	        // ----------------------------------------->>>>>>> STATUS MANUAL <<<<<<<-----------------------------------------
	        
	        // Write to static from IO
	        // ACTIVATE --> MANUAL MODE
	        // ProductionLine
	        IF #Active.Line.ProductionLine THEN
	            // SET --> MANUAL MODE
	            IF DB_Manual.Line.ProductionLine.Conveyor[#ConveyorID].ManualEnable THEN
	                #ReadConveyorStatus.Manual := TRUE;
	            END_IF;
	            // RESET --> MANUAL MODE
	            IF NOT DB_Manual.Line.ProductionLine.Conveyor[#ConveyorID].ManualEnable AND #SSR.ResetSystem THEN
	                #ReadConveyorStatus.Manual := FALSE;
	            END_IF;
	        END_IF;
	        // EmptyLine
	        IF #Active.Line.EmptyLine THEN
	            // SET --> MANUAL MODE
	            IF DB_Manual.Line.EmptyLine.Conveyor[#ConveyorID].ManualEnable THEN
	                #ReadConveyorStatus.Manual := TRUE;
	            END_IF;
	            // RESET --> MANUAL MODE
	            IF NOT DB_Manual.Line.EmptyLine.Conveyor[#ConveyorID].ManualEnable AND #SSR.ResetSystem THEN
	                #ReadConveyorStatus.Manual := FALSE;
	            END_IF;
	        END_IF;
	        // PackedLine
	        IF #Active.Line.PackedLine THEN
	            // SET --> MANUAL MODE
	            IF DB_Manual.Line.PackedLine.Conveyor[#ConveyorID].ManualEnable THEN
	                #ReadConveyorStatus.Manual := TRUE;
	            END_IF;
	            // RESET --> MANUAL MODE
	            IF NOT DB_Manual.Line.PackedLine.Conveyor[#ConveyorID].ManualEnable AND #SSR.ResetSystem THEN
	                #ReadConveyorStatus.Manual := FALSE;
	            END_IF;
	        END_IF;
	        
	        // Manual enable and Run from HMI
	        // ProductionLine
	        IF #Active.Line.ProductionLine THEN
	            IF #ConveyorID = DB_Manual.Conveyor.ID THEN
	                DB_Manual.Line.ProductionLine.Conveyor[DB_Manual.Conveyor.ID].ManualEnable := DB_Manual.Conveyor.Enable;
	                DB_Manual.Line.ProductionLine.Conveyor[DB_Manual.Conveyor.ID].Run.Forward := DB_Manual.Conveyor.in;
	            END_IF;
	        END_IF;
	        // EmptyLine
	        IF #Active.Line.EmptyLine THEN
	            IF #ConveyorID = DB_Manual.Conveyor.ID THEN
	                DB_Manual.Line.EmptyLine.Conveyor[DB_Manual.Conveyor.ID].ManualEnable := DB_Manual.Conveyor.Enable;
	                DB_Manual.Line.EmptyLine.Conveyor[DB_Manual.Conveyor.ID].Run.Forward := DB_Manual.Conveyor.in;
	            END_IF;
	        END_IF;
	        // PackedLine
	        IF #Active.Line.PackedLine THEN
	            IF #ConveyorID = DB_Manual.Conveyor.ID THEN
	                DB_Manual.Line.PackedLine.Conveyor[DB_Manual.Conveyor.ID].ManualEnable := DB_Manual.Conveyor.Enable;
	                DB_Manual.Line.PackedLine.Conveyor[DB_Manual.Conveyor.ID].Run.Forward := DB_Manual.Conveyor.in;
	            END_IF;
	        END_IF;
	        
	    END_REGION
	    
	    REGION Status Stop
	        
	        // ----------------------------------------->>>>>>> STATUS STOP <<<<<<<-----------------------------------------
	        
	        IF #SSR.StopSystem THEN
	            #ReadConveyorStatus.Stop := TRUE;
	        END_IF;
	        IF #SSR.StartSystem OR #SSR.ResetSystem THEN
	            #ReadConveyorStatus.Stop := FALSE;
	        END_IF;
	        
	    END_REGION
	    
	    REGION Sensor Blockage
	        
	        // ----------------------------------------->>>>>>> STATUS BLOCKAGE <<<<<<<------------------------------------
	        
	        // FB_SensorBlockage
	        // called as MIDB
	        #CONVEYOR_SENSOR_BLOCKAGE(ConveyorSensor       := #FilteredSensor,
	                                  StatusRunning        := #ReadConveyorStatus.Running,
	                                  SensorBlockagePeriod := #ReadConveyorParameters.SensorBlockageTime,
	                                  SensorBlocked        => #ConveyorFault.Sensor_Blockage,
	                                  ReadBlockageStatus   => #ReadConveyorStatus.Blockage);
	        
	        REGION alarm 
	            
	            // ==========================
	            // Sensor Blockage: HMI Alarm
	            // ==========================
	            // Sensor blockage alarm message is written to the alarm word
	            // corresponding to the active line
	            // ProductionLine
	            IF #Active.Line.ProductionLine THEN
	                DB_Alarm."word".Line.ProductionLine.Conveyor[#ConveyorID].%X0 := #ReadConveyorStatus.Blockage;
	            END_IF;
	            // EmptyLine
	            IF #Active.Line.EmptyLine THEN
	                DB_Alarm."word".Line.EmptyLine.Conveyor[#ConveyorID].%X0 := #ReadConveyorStatus.Blockage;
	            END_IF;
	            // PackedLine
	            IF #Active.Line.PackedLine THEN
	                DB_Alarm."word".Line.PackedLine.Conveyor[#ConveyorID].%X0 := #ReadConveyorStatus.Blockage;
	            END_IF;
	            
	        END_REGION
	        
	    END_REGION
	    
	    REGION Visu Color
	        
	        // each and every status of the conveyor will be mentioned by different colors in HMI panel
	        
	        #VisuColor.%X8 := #ReadConveyorStatus.Blockage;
	        #VisuColor.%X0 := #ReadConveyorStatus.ON;
	        #VisuColor.%X1 := #ReadConveyorStatus.ReadytoRun;
	        #VisuColor.%X2 := #ReadConveyorStatus.Occupied;
	        #VisuColor.%X3 := #ReadConveyorStatus.Running;
	        #VisuColor.%X4 := #ReadConveyorStatus.Fault;
	        #VisuColor.%X5 := #ReadConveyorStatus.Estop;
	        #VisuColor.%X6 := #ReadConveyorStatus.Manual;
	        #VisuColor.%X7 := #ReadConveyorStatus.Stop;
	        
	        // convert word to Interger value: 
	        // color will be depends on the status priority (integer value) 
	        // reference: Conveyor image in HMI screen -> property -> Apperance   
	        
	        // ProductionLine
	        IF #Active.Line.ProductionLine THEN
	            DB_VisuColor.Line.ProductionLine.Conveyor[#ConveyorID] :=
	            WORD_TO_INT(#VisuColor);
	        END_IF;
	        // EmptyLine
	        IF #Active.Line.EmptyLine THEN
	            DB_VisuColor.Line.EmptyLine.Conveyor[#ConveyorID] :=
	            WORD_TO_INT(#VisuColor);
	        END_IF;
	        // PackedLine
	        IF #Active.Line.PackedLine THEN
	            DB_VisuColor.Line.PackedLine.Conveyor[#ConveyorID] :=
	            WORD_TO_INT(#VisuColor);
	        END_IF;
	        
	    END_REGION
	    
	    REGION Global Status
	        
	        // write -> global status
	        // ProductionLine
	        IF #Active.Line.ProductionLine THEN
	            DB_Global.Status.Line.ProductionLine.On[#ConveyorID] := #ReadConveyorStatus.ON;
	            DB_Global.Status.Line.ProductionLine.ReadyToRun[#ConveyorID] := #ReadConveyorStatus.ReadytoRun;
	            DB_Global.Status.Line.ProductionLine.Occupied[#ConveyorID] := #ReadConveyorStatus.Occupied;
	            DB_Global.Status.Line.ProductionLine.Running[#ConveyorID] := #ReadConveyorStatus.Running;
	            DB_Global.Status.Line.ProductionLine.Fault[#ConveyorID] := #ReadConveyorStatus.Fault;
	            DB_Global.Status.Line.ProductionLine.Estop[#ConveyorID] := #ReadConveyorStatus.Estop;
	            DB_Global.Status.Line.ProductionLine.Manual[#ConveyorID] := #ReadConveyorStatus.Manual;
	            DB_Global.Status.Line.ProductionLine.Stop[#ConveyorID] := #ReadConveyorStatus.Stop;
	            DB_Global.Status.Line.ProductionLine.Blockage[#ConveyorID] := #ReadConveyorStatus.Blockage;
	        END_IF;
	        // EmptyLine
	        IF #Active.Line.EmptyLine THEN
	            DB_Global.Status.Line.EmptyLine.On[#ConveyorID] := #ReadConveyorStatus.ON;
	            DB_Global.Status.Line.EmptyLine.ReadyToRun[#ConveyorID] := #ReadConveyorStatus.ReadytoRun;
	            DB_Global.Status.Line.EmptyLine.Occupied[#ConveyorID] := #ReadConveyorStatus.Occupied;
	            DB_Global.Status.Line.EmptyLine.Running[#ConveyorID] := #ReadConveyorStatus.Running;
	            DB_Global.Status.Line.EmptyLine.Fault[#ConveyorID] := #ReadConveyorStatus.Fault;
	            DB_Global.Status.Line.EmptyLine.Estop[#ConveyorID] := #ReadConveyorStatus.Estop;
	            DB_Global.Status.Line.EmptyLine.Manual[#ConveyorID] := #ReadConveyorStatus.Manual;
	            DB_Global.Status.Line.EmptyLine.Stop[#ConveyorID] := #ReadConveyorStatus.Stop;
	            DB_Global.Status.Line.EmptyLine.Blockage[#ConveyorID] := #ReadConveyorStatus.Blockage;
	        END_IF;
	        // PackedLine
	        IF #Active.Line.PackedLine THEN
	            DB_Global.Status.Line.PackedLine.On[#ConveyorID] := #ReadConveyorStatus.ON;
	            DB_Global.Status.Line.PackedLine.ReadyToRun[#ConveyorID] := #ReadConveyorStatus.ReadytoRun;
	            DB_Global.Status.Line.PackedLine.Occupied[#ConveyorID] := #ReadConveyorStatus.Occupied;
	            DB_Global.Status.Line.PackedLine.Running[#ConveyorID] := #ReadConveyorStatus.Running;
	            DB_Global.Status.Line.PackedLine.Fault[#ConveyorID] := #ReadConveyorStatus.Fault;
	            DB_Global.Status.Line.PackedLine.Estop[#ConveyorID] := #ReadConveyorStatus.Estop;
	            DB_Global.Status.Line.PackedLine.Manual[#ConveyorID] := #ReadConveyorStatus.Manual;
	            DB_Global.Status.Line.PackedLine.Stop[#ConveyorID] := #ReadConveyorStatus.Stop;
	            DB_Global.Status.Line.PackedLine.Blockage[#ConveyorID] := #ReadConveyorStatus.Blockage;
	        END_IF;
	        
	    END_REGION
	    
	END_REGION
	
	REGION Run/Stop Conveyor 
	    
	    // FB_ConveyorRunStop
	    // Called as MIDB
	    
	    #"RUN/STOP_CONVEYOR"(StatusReady  := #ReadConveyorStatus.ReadytoRun,
	                         StatusOccu   := #ReadConveyorStatus.Occupied,
	                         DSOcc        := #Downstream,
	                         USOcc        := #Upstream,
	                         EnergySave   := #EnergySave,
	                         ILStop       := #Interlock,
	                         PecBlockage  := #ConveyorFault.Sensor_Blockage,
	                         MotorForward => #StartMotorForward,
	                         MotorReverse => #StartMotorReverse);
	    
	END_REGION
	
	REGION Energy Save
	    
	    // FB_EnergySave
	    // Called as MIDB
	    
	    #ENERGY_SAVE(StatusReady      := #ReadConveyorStatus.ReadytoRun,
	                 StatusOccupied   := #ReadConveyorStatus.Occupied,
	                 StartUpIN        := #SetStartUp,
	                 USOcc            := #Upstream,
	                 EnergySaveTimePT := #ReadConveyorParameters.EnergySaveTime,
	                 EnergySaveOut    => #EnergySave);
	    
	END_REGION
	
	REGION Write logic and parameters
	    
	    // Motor Forward: motors which has only one control bit
	    // ProductionLine 
	    IF #Active.Line.ProductionLine THEN
	        #RunForward :=
	        (#StartMotorForward AND NOT #StartMotorReverse) // Automatic mode
	        OR (#ReadConveyorStatus.Manual AND DB_Manual.Line.ProductionLine.Conveyor[#ConveyorID].Run.Forward); //Manual mode
	    END_IF;
	    // EmptyLine 
	    IF #Active.Line.EmptyLine THEN
	        #RunForward :=
	        (#StartMotorForward AND NOT #StartMotorReverse) // Automatic mode
	        OR (#ReadConveyorStatus.Manual AND DB_Manual.Line.EmptyLine.Conveyor[#ConveyorID].Run.Forward); //Manual mode
	    END_IF;
	    // PackedLine 
	    IF #Active.Line.PackedLine THEN
	        #RunForward :=
	        (#StartMotorForward AND NOT #StartMotorReverse) // Automatic mode
	        OR (#ReadConveyorStatus.Manual AND DB_Manual.Line.PackedLine.Conveyor[#ConveyorID].Run.Forward); //Manual mode
	    END_IF;
	    
	    REGION Bihl Wiedemann 
	        
	        // process data for BW-ASi
	        
	        IF #MotorType."24v-ASi" THEN
	            
	            REGION Direction
	                
	                // ProductionLine
	                IF #Active.Line.ProductionLine THEN
	                    #WriteAsiDir := DB_AsiSetpoint.Line.ProductionLine.DirChange.Conveyor[#ConveyorID];
	                END_IF;
	                // EmptyLine
	                IF #Active.Line.EmptyLine THEN
	                    #WriteAsiDir := DB_AsiSetpoint.Line.EmptyLine.DirChange.Conveyor[#ConveyorID];
	                END_IF;
	                // PackedLine
	                IF #Active.Line.PackedLine THEN
	                    #WriteAsiDir := DB_AsiSetpoint.Line.PackedLine.DirChange.Conveyor[#ConveyorID];
	                END_IF;
	                
	            END_REGION
	            
	            REGION Speed
	                
	                // ProductionLine
	                IF #Active.Line.ProductionLine THEN
	                    #WriteAsiSpeed := DB_AsiSetpoint.Line.ProductionLine.Speed.Conveyor[#ConveyorID];
	                END_IF;
	                // EmptyLine
	                IF #Active.Line.EmptyLine THEN
	                    #WriteAsiSpeed := DB_AsiSetpoint.Line.EmptyLine.Speed.Conveyor[#ConveyorID];
	                END_IF;
	                // PackedLine
	                IF #Active.Line.PackedLine THEN
	                    #WriteAsiSpeed := DB_AsiSetpoint.Line.PackedLine.Speed.Conveyor[#ConveyorID];
	                END_IF;
	                
	            END_REGION
	            
	        END_IF;
	        
	    END_REGION
	    
	    REGION NORD (Line shaft)
	        
	        // process data and logic for NORD VFD
	        
	        IF #MotorType.nord THEN
	            
	            // ProductionLine
	            IF #Active.Line.ProductionLine THEN
	                
	                IF NOT #ReadConveyorStatus.Fault THEN
	                    IF // Nord Motor Run - Automatic mode
	                        ((#ReadConveyorStatus.ReadytoRun AND
	                        #StartMotorForward) OR
	                        // Nord Motor Run - manual mode
	                        (#ReadConveyorStatus.Manual AND
	                        DB_Manual.Line.ProductionLine.Conveyor[#ConveyorID].Run.Forward))
	                    THEN
	                        #NordControlEnable := #NordSetpointRun;
	                    ELSE
	                        #NordControlEnable := #NordSetpointReady;
	                    END_IF;
	                END_IF;
	                
	                // Nord Motor Fault ack
	                IF #ReadConveyorStatus.Fault AND #SSR.ResetSystem THEN
	                    #NordControlEnable := #NordFaultAck;
	                END_IF;
	                
	                // Nord setpoint
	                #NordSetpoint := DINT_TO_WORD(DB_NordSetPoint.Line.ProductionLine.Conveyor[#ConveyorID]);
	                
	            END_IF;
	            
	            // EmptyLine
	            IF #Active.Line.EmptyLine THEN
	                
	                IF NOT #ReadConveyorStatus.Fault THEN
	                    IF // Nord Motor Run - Automatic mode
	                        ((#ReadConveyorStatus.ReadytoRun AND
	                        #StartMotorForward) OR
	                        // Nord Motor Run - manual mode
	                        (#ReadConveyorStatus.Manual AND
	                        DB_Manual.Line.EmptyLine.Conveyor[#ConveyorID].Run.Forward))
	                    THEN
	                        #NordControlEnable := #NordSetpointRun;
	                    ELSE
	                        #NordControlEnable := #NordSetpointReady;
	                    END_IF;
	                END_IF;
	                
	                // Nord Motor Fault ack
	                IF #ReadConveyorStatus.Fault AND #SSR.ResetSystem THEN
	                    #NordControlEnable := #NordFaultAck;
	                END_IF;
	                
	                // Nord setpoint
	                #NordSetpoint := DINT_TO_WORD(DB_NordSetPoint.Line.EmptyLine.Conveyor[#ConveyorID]);
	                
	            END_IF;
	            
	            // PackedLine
	            IF #Active.Line.PackedLine THEN
	                
	                IF NOT #ReadConveyorStatus.Fault THEN
	                    IF // Nord Motor Run - Automatic mode
	                        ((#ReadConveyorStatus.ReadytoRun AND
	                        #StartMotorForward) OR
	                        // Nord Motor Run - manual mode
	                        (#ReadConveyorStatus.Manual AND
	                        DB_Manual.Line.PackedLine.Conveyor[#ConveyorID].Run.Forward))
	                    THEN
	                        #NordControlEnable := #NordSetpointRun;
	                    ELSE
	                        #NordControlEnable := #NordSetpointReady;
	                    END_IF;
	                END_IF;
	                
	                // Nord Motor Fault ack
	                IF #ReadConveyorStatus.Fault AND #SSR.ResetSystem THEN
	                    #NordControlEnable := #NordFaultAck;
	                END_IF;
	                
	                // Nord setpoint
	                #NordSetpoint := DINT_TO_WORD(DB_NordSetPoint.Line.PackedLine.Conveyor[#ConveyorID]);
	                
	            END_IF;
	            
	            
	   END_IF;
	            
	            
	END_REGION
	
	REGION Interroll Multi control roller
	    
	    // process data for Interroll multicontrol card
	    IF #MotorType."24v-IMC" THEN
	    // PackedLine
	        IF #Active.Line.PackedLine THEN
	            IF (#StartMotorForward AND NOT #StartMotorReverse)
	            OR (#ReadConveyorStatus.Manual AND
	            DB_Manual.Line.PackedLine.Conveyor[#ConveyorID].Run.Forward AND
	            NOT DB_Manual.Line.PackedLine.Conveyor[#ConveyorID].Run.Reverse)
	           THEN
	            #ImcSpeed := #ReadConveyorParameters."IMC-SpeedSetPoint";
	           ELSE
	            #ImcSpeed := #NullSpeed;
	           END_IF;
	       END_IF;
	   END_IF;
	   
	END_REGION
	    
	END_REGION
	
END_FUNCTION_BLOCK
END_NAMESPACE

NAMESPACE Global
FUNCTION_BLOCK FB_MABS
{ S7_Optimized_Access := 'TRUE' ; Published := 'TRUE' }
VERSION : 0.1
   VAR_INPUT 
      MABS_ID : Int;
      CrossSensor : Bool;
      ErrorSignal : Bool;
      Upstream : Bool;
      UpstreamRunning : Bool;
      Downstream_Straight : Bool;
      "Downstream_Right/Left" : Bool;
      SortDir : ItemDir;
      RemoteOut1 : Bool;
      RemoteOut2 : Bool;
      RemoteOut3 : Bool;
      RemoteOut4 : Bool;
      Parameter : MABS_Parameters;
   END_VAR

   VAR_OUTPUT 
      RemoteIn1 : Bool;
      RemoteIn2 : Bool;
      RemoteIn3 : Bool;
      RunWheels : Bool;
   END_VAR

   VAR 
      ReadInputSignal : Struct
         CrossSensor : Bool;
         EmergencyStop : Bool;
         ErrorSignal : Bool;
      END_STRUCT;
      Active : Struct
         Line : Struct
            ProductionLine : Bool;
            EmptyLine : Bool;
            PackedLine : Bool;
         END_STRUCT;
         EstopZone { S7_SetPoint := 'False'} : EsopZone;
      END_STRUCT;
      CROSS_SENSOR_FILTER { S7_SetPoint := 'False'} : FB_Sensor;
      MABS_SENSOR_BLOCKAGE {InstructionName := 'IEC_TIMER'; LibVersion := '1.0'} : IEC_TIMER;
      MABS_STATUS_ON { S7_SetPoint := 'False'} : FB_StatusON;
      MABS_STATUS_READY { S7_SetPoint := 'False'} : FB_StatusReady;
      MABS_STATUS_FAULT { S7_SetPoint := 'False'} : FB_StatusFault;
      AUTO_RESET { S7_SetPoint := 'False'} : FB_AutoReset;
      SSR { S7_SetPoint := 'False'} : SystemSSR;
      ReadMabsStatus { S7_SetPoint := 'False'} : ConveyorStatus;
      MABSFault { S7_SetPoint := 'False'} : Fault;
      SimuMode : Struct
         Sensor : Bool;
         Fault : Bool;
      END_STRUCT;
      StartUpTimer {InstructionName := 'TOF_TIME'; LibVersion := '1.0'; S7_SetPoint := 'False'} : TOF_TIME;
      FT_StartUp {InstructionName := 'F_TRIG'; LibVersion := '1.0'} : F_TRIG;
      SetStartUp { S7_SetPoint := 'True'} : Bool;
      VisuColor : Word;
      PhaseError : Bool;
      StartupMABS { S7_SetPoint := 'True'} : Bool;
      FilteredSensor { S7_SetPoint := 'True'} : Bool;
      AutoReset { S7_SetPoint := 'True'} : Bool;
      StopSystemFireActive : Bool;
      Sort { S7_SetPoint := 'False'} : ItemDir;
      mabs : Struct
         RemoteIn1 : Bool;
         RemoteIn2 : Bool;
         RemoteIn3 : Bool;
         RemoteIn4 : Bool;
         Wheels : Bool;
      END_STRUCT;
      Home : Bool;
      HomeCheckTimer {InstructionName := 'TON_TIME'; LibVersion := '1.0'} : TON_TIME;
      CurrentPosition : Struct
         left : Bool;
         right : Bool;
         straight : Bool;
      END_STRUCT;
      RT_DelaySwing_Straight {InstructionName := 'R_TRIG'; LibVersion := '1.0'} : R_TRIG;
      RT_DelaySwing_toRight {InstructionName := 'R_TRIG'; LibVersion := '1.0'} : R_TRIG;
      RT_DelaySwing_toLeft {InstructionName := 'R_TRIG'; LibVersion := '1.0'} : R_TRIG;
      ToSt_DelayTimer {InstructionName := 'TON_TIME'; LibVersion := '1.0'} : TON_TIME;
      ToRt_DelayTimer {InstructionName := 'TON_TIME'; LibVersion := '1.0'} : TON_TIME;
      ToLt_DelayTimer {InstructionName := 'TON_TIME'; LibVersion := '1.0'} : TON_TIME;
      St_SwingDelay { S7_SetPoint := 'True'} : Bool;
      Rt_SwingDelay : Bool;
      Lt_SwingDelay : Bool;
      noSwing : Bool;
      CmdExFailure : Struct
         "Timer" {InstructionName := 'TONR_TIME'; LibVersion := '1.0'} : TONR_TIME;
         UpstreamCheckTimer {InstructionName := 'TONR_TIME'; LibVersion := '1.0'} : TONR_TIME;
      END_STRUCT;
      FT_Upstream {InstructionName := 'F_TRIG'; LibVersion := '1.0'; S7_SetPoint := 'False'} : F_TRIG;
      RT_DS_St {InstructionName := 'R_TRIG'; LibVersion := '1.0'} : R_TRIG;
      "RT_DS_Rt/Lt" {InstructionName := 'R_TRIG'; LibVersion := '1.0'} : R_TRIG;
      RT_ToStraight {InstructionName := 'R_TRIG'; LibVersion := '1.0'; S7_SetPoint := 'False'} : R_TRIG;
      RT_ToRight {InstructionName := 'R_TRIG'; LibVersion := '1.0'} : R_TRIG;
      RT_ToLeft {InstructionName := 'R_TRIG'; LibVersion := '1.0'} : R_TRIG;
      FT_Blockage {InstructionName := 'F_TRIG'; LibVersion := '1.0'} : F_TRIG;
      HoldFailure { S7_SetPoint := 'True'} : Bool;
      MABS_Wheel {InstructionName := 'TOF_TIME'; LibVersion := '1.0'; S7_SetPoint := 'False'} : TOF_TIME;
      RT_Sort_St {InstructionName := 'R_TRIG'; LibVersion := '1.0'} : R_TRIG;
      RT_Sort_Rt {InstructionName := 'R_TRIG'; LibVersion := '1.0'} : R_TRIG;
      RT_Sort_Lt {InstructionName := 'R_TRIG'; LibVersion := '1.0'} : R_TRIG;
      HoldSwingTimer {InstructionName := 'TOF_TIME'; LibVersion := '1.0'} : TOF_TIME;
      HoldSwing { S7_SetPoint := 'True'} : Bool;
   END_VAR


BEGIN
	// ==========================================================================================================================================
	// Company        : LogTech, s.r.o.
	// Created by     : Anton Vinoth Soundraraj
	// Block          : FB_MABS
	// Project        : Lékarna DC Chrudim
	// Project number : 23-157
	// ==========================================================================================================================================
	
	REGION Active Line
	    
	    // ProductionLine
	    IF (#MABS_ID >= _.gminProductionLine AND
	        #MABS_ID <= _.gmaxProductionLine)
	    THEN
	        #Active.Line.ProductionLine := TRUE;
	    END_IF;
	    
	    // EmptyLine
	    IF (#MABS_ID >= _.gminEmptyLine AND
	        #MABS_ID <= _.gmaxEmptyLine)
	    THEN
	        #Active.Line.EmptyLine := TRUE;
	    END_IF;
	    
	    // PackedLine
	    IF (#MABS_ID >= _.gminPackedLine AND
	        #MABS_ID <= _.gmaxPackedLine)
	    THEN
	        #Active.Line.PackedLine := TRUE;
	    END_IF;
	    
	END_REGION
	    
	
	REGION Estop zone
	    
	    // Production Line A1
	    IF (#MABS_ID >= _."gA1.6.1" AND
	        #MABS_ID <= _."gA1.6.2") OR
	        // Empty Line A1
	        (#MABS_ID >= _."gJ1.5.2" AND
	        #MABS_ID <= _."gJ1.6.2")
	    THEN
	        #Active.EstopZone."1" := TRUE;
	    END_IF;
	    
	    // Production Line A2
	    IF (#MABS_ID >= _."gA1.9.1" AND
	        #MABS_ID <= _."gA1.9.2")
	    THEN
	        #Active.EstopZone."2" := TRUE;
	    END_IF;
	    
	END_REGION
	
	REGION Read Simu inputs  
	    
	    // ProductionLine
	    IF #Active.Line.ProductionLine THEN
	        // read simu
	        #SimuMode.Sensor := DB_SystemSimu.TriggerSensor.Line.ProductionLine.Conveyor[#MABS_ID];
	        #SimuMode.Fault := DB_SystemSimu.TriggerFault.Line.ProductionLine.Conveyor[#MABS_ID];
	    END_IF;
	    
	    // EmptyLine
	    IF #Active.Line.EmptyLine THEN
	        // read simu
	        #SimuMode.Sensor := DB_SystemSimu.TriggerSensor.Line.EmptyLine.Conveyor[#MABS_ID];
	        #SimuMode.Fault := DB_SystemSimu.TriggerFault.Line.EmptyLine.Conveyor[#MABS_ID];
	    END_IF;
	    
	    // PackedLine
	    IF #Active.Line.PackedLine THEN
	        // read simu
	        #SimuMode.Sensor := DB_SystemSimu.TriggerSensor.Line.PackedLine.Conveyor[#MABS_ID];
	        #SimuMode.Fault := DB_SystemSimu.TriggerFault.Line.PackedLine.Conveyor[#MABS_ID];
	    END_IF;
	    
	END_REGION
	
	REGION SystemSSR
	    
	    //Zone 1
	    IF #Active.EstopZone."1" THEN
	        #SSR.StartSystem := DB_SystemSSR.Zone."1".StartSystem;
	        #SSR.StopSystem := DB_SystemSSR.Zone."1".StopSystem;
	        #SSR.ResetSystem := DB_SystemSSR.Zone."1".ResetSystem;
	    END_IF;
	    
	    //Zone 2
	    IF #Active.EstopZone."2" THEN
	        #SSR.StartSystem := DB_SystemSSR.Zone."2".StartSystem;
	        #SSR.StopSystem := DB_SystemSSR.Zone."2".StopSystem;
	        #SSR.ResetSystem := DB_SystemSSR.Zone."2".ResetSystem;
	    END_IF;
	    
	END_REGION
	
	REGION Read Input
	    
	    // read all inputs to the block
	    // Conveyor input read signals
	    #ReadInputSignal.CrossSensor := #CrossSensor OR
	    #SimuMode.Sensor; // simu call
	    #ReadInputSignal.ErrorSignal := #ErrorSignal OR
	    #SimuMode.Fault; // simu call;
	    // estop
	    #ReadInputSignal.EmergencyStop := _.DB_SafetyStandard.ToStandard.EstopActive;
	    
	END_REGION
	
	REGION Conveyor startup
	    
	    // Conveyor StartUp: Conveyor startup signal after 5 second delay
	    
	    #StartUpTimer.TOF(IN := #SSR.StartSystem,
	                      PT := #Parameter.StartUpTime);
	    
	    #FT_StartUp(CLK := #StartUpTimer.Q);
	    
	    // set startup after 5 seconds
	    #SetStartUp := #FT_StartUp.Q;
	    
	END_REGION
	
	REGION READ AND INIT
	    
	    REGION FIRE
	        
	        // Fire signal from fire system stops the whole system
	        // System can be reset from Fire status only if the fire signal is deactivated
	        
	        // FIRE ALARM ACTIVE --> STOP SYSTEM
	        IF DB_SystemSimu.Fire THEN
	            #StopSystemFireActive := TRUE;
	        END_IF;
	        // RESET --> FIRE ALARM
	        IF #SSR.ResetSystem AND NOT DB_SystemSimu.Fire THEN
	            #StopSystemFireActive := FALSE;
	        END_IF;
	        
	    END_REGION
	    
	END_REGION
	
	REGION Conveyor Status
	    
	    REGION Status ON
	        
	        // ----------------------------------------->>>>>>> STATUS ON <<<<<<<-----------------------------------------
	        // FB_ConveyorStatusON
	        // called as IDMB
	        
	        #MABS_STATUS_ON(SystemStartActive := #SSR.StartSystem,
	                        StatusStop := #ReadMabsStatus.Stop,
	                        StatusEStop := #ReadMabsStatus.Estop,
	                        StatusManual := #ReadMabsStatus.Manual,
	                        StatusFault := #ReadMabsStatus.Fault,
	                        FireAlarmActive := #StopSystemFireActive,
	                        StatusON => #ReadMabsStatus.ON);
	        
	    END_REGION
	    
	    REGION Status Ready
	        
	        // ----------------------------------------->>>>>>> STATUS READY <<<<<<<-----------------------------------------
	        // FB_ConveyorStatusReady
	        // called as MIDB
	        
	        #MABS_STATUS_READY(StatusON := #ReadMabsStatus.ON,
	                           StatusESTOP := #ReadMabsStatus.Estop,
	                           StatusFAULT := #ReadMabsStatus.Fault,
	                           StatusMAN := #ReadMabsStatus.Manual,
	                           SignalFIRE := #StopSystemFireActive,
	                           SystemAlertTime := #Parameter.StartUpTime,
	                           StatusReady => #ReadMabsStatus.ReadytoRun);
	        
	    END_REGION
	    
	    REGION Status Occupied
	        
	        // ----------------------------------------->>>>>>> STATUS OCCUPIED <<<<<<<-----------------------------------------
	        
	        #ReadMabsStatus.Occupied :=
	        #CROSS_SENSOR_FILTER.FilteredSensor;
	        
	    END_REGION
	    
	    REGION Status Running
	        
	        // ----------------------------------------->>>>>>> STATUS RUNNING <<<<<<<-----------------------------------------
	        
	        #ReadMabsStatus.Running :=
	        #ReadMabsStatus.ReadytoRun AND
	        #mabs.Wheels;
	        
	    END_REGION
	    
	    REGION Status Fault
	        
	        // ----------------------------------------->>>>>>> STATUS FAULT <<<<<<<-----------------------------------------
	        
	        // Reading error signal from the motor drive
	        #MABSFault.Motor_Error := #ReadInputSignal.ErrorSignal;
	        
	        // FC_ConveyorStatusFault
	        #MABS_STATUS_FAULT(FaultActive := #MABSFault.Motor_Error,
	                           ResetFault := #SSR.ResetSystem,
	                           StatusRunning := #ReadMabsStatus.Running,
	                           FaultStatus => #ReadMabsStatus.Fault);
	        
	    END_REGION
	    
	    REGION Status ESTOP
	        
	        // ----------------------------------------->>>>>>> STATUS ESTOP <<<<<<<-----------------------------------------
	        
	        #AUTO_RESET(AckIN := #SSR.ResetSystem,
	                    Ack => #AutoReset);
	        
	        // EMERGENCY STOP ACTIVE --> STOP SYSTEM
	        IF #ReadInputSignal.EmergencyStop THEN
	            #ReadMabsStatus.Estop := TRUE;
	        END_IF;
	        // RESET --> EMERGENCY STOP
	        IF #AutoReset AND NOT #ReadInputSignal.EmergencyStop THEN
	            #ReadMabsStatus.Estop := FALSE;
	        END_IF;
	        
	    END_REGION
	    
	    REGION Status Stop
	        
	        // ----------------------------------------->>>>>>> STATUS STOP <<<<<<<-----------------------------------------
	        
	        IF #SSR.StopSystem THEN
	            #ReadMabsStatus.Stop := TRUE;
	        END_IF;
	        IF #SSR.StartSystem OR #SSR.ResetSystem THEN
	            #ReadMabsStatus.Stop := FALSE;
	        END_IF;
	        
	    END_REGION
	    
	    REGION Sensor Blockage
	        
	        // ----------------------------------------->>>>>>> STATUS BLOCKAGE <<<<<<<-------------------------------------
	        
	        // FB_SensorBlockage
	        // called as MIDB
	        
	        #MABS_SENSOR_BLOCKAGE.TON(IN := #ReadMabsStatus.ReadytoRun AND
	                                  #CROSS_SENSOR_FILTER.FilteredSensor,
	                                  PT := #Parameter.SensorBlockageTime,
	                                  Q => #ReadMabsStatus.Blockage);
	        
	        // ==========================
	        // Sensor Blockage: HMI Alarm
	        // ==========================
	        // Sensor blockage alarm message is written to the first bit of the alarm word
	        // corresponding to the active line
	        
	        REGION alarm 
	            
	            // ==========================
	            // Sensor Blockage: HMI Alarm
	            // ==========================
	            // Sensor blockage alarm message is written to the alarm word
	            // corresponding to the active line
	            // ProductionLine
	            IF #Active.Line.ProductionLine THEN
	                DB_Alarm."word".Line.ProductionLine.Conveyor[#MABS_ID].%X0 := #ReadMabsStatus.Blockage;
	            END_IF;
	            // EmptyLine
	            IF #Active.Line.EmptyLine THEN
	                DB_Alarm."word".Line.EmptyLine.Conveyor[#MABS_ID].%X0 := #ReadMabsStatus.Blockage;
	            END_IF;
	            // PackedLine
	            IF #Active.Line.PackedLine THEN
	                DB_Alarm."word".Line.PackedLine.Conveyor[#MABS_ID].%X0 := #ReadMabsStatus.Blockage;
	            END_IF;
	            
	        END_REGION
	        
	    END_REGION
	    
	    REGION Global Status
	        
	        // write -> global status
	        // ProductionLine
	        IF #Active.Line.ProductionLine THEN
	            DB_Global.Status.Line.ProductionLine.On[#MABS_ID] := #ReadMabsStatus.ON;
	            DB_Global.Status.Line.ProductionLine.ReadyToRun[#MABS_ID] := #ReadMabsStatus.ReadytoRun;
	            DB_Global.Status.Line.ProductionLine.Occupied[#MABS_ID] := #ReadMabsStatus.Occupied;
	            DB_Global.Status.Line.ProductionLine.Running[#MABS_ID] := #ReadMabsStatus.Running;
	            DB_Global.Status.Line.ProductionLine.Fault[#MABS_ID] := #ReadMabsStatus.Fault;
	            DB_Global.Status.Line.ProductionLine.Estop[#MABS_ID] := #ReadMabsStatus.Estop;
	            DB_Global.Status.Line.ProductionLine.Manual[#MABS_ID] := #ReadMabsStatus.Manual;
	            DB_Global.Status.Line.ProductionLine.Stop[#MABS_ID] := #ReadMabsStatus.Stop;
	            DB_Global.Status.Line.ProductionLine.Blockage[#MABS_ID] := #ReadMabsStatus.Blockage;
	        END_IF;
	        // EmptyLine
	        IF #Active.Line.EmptyLine THEN
	            DB_Global.Status.Line.EmptyLine.On[#MABS_ID] := #ReadMabsStatus.ON;
	            DB_Global.Status.Line.EmptyLine.ReadyToRun[#MABS_ID] := #ReadMabsStatus.ReadytoRun;
	            DB_Global.Status.Line.EmptyLine.Occupied[#MABS_ID] := #ReadMabsStatus.Occupied;
	            DB_Global.Status.Line.EmptyLine.Running[#MABS_ID] := #ReadMabsStatus.Running;
	            DB_Global.Status.Line.EmptyLine.Fault[#MABS_ID] := #ReadMabsStatus.Fault;
	            DB_Global.Status.Line.EmptyLine.Estop[#MABS_ID] := #ReadMabsStatus.Estop;
	            DB_Global.Status.Line.EmptyLine.Manual[#MABS_ID] := #ReadMabsStatus.Manual;
	            DB_Global.Status.Line.EmptyLine.Stop[#MABS_ID] := #ReadMabsStatus.Stop;
	            DB_Global.Status.Line.EmptyLine.Blockage[#MABS_ID] := #ReadMabsStatus.Blockage;
	        END_IF;
	        // PackedLine
	        IF #Active.Line.PackedLine THEN
	            DB_Global.Status.Line.PackedLine.On[#MABS_ID] := #ReadMabsStatus.ON;
	            DB_Global.Status.Line.PackedLine.ReadyToRun[#MABS_ID] := #ReadMabsStatus.ReadytoRun;
	            DB_Global.Status.Line.PackedLine.Occupied[#MABS_ID] := #ReadMabsStatus.Occupied;
	            DB_Global.Status.Line.PackedLine.Running[#MABS_ID] := #ReadMabsStatus.Running;
	            DB_Global.Status.Line.PackedLine.Fault[#MABS_ID] := #ReadMabsStatus.Fault;
	            DB_Global.Status.Line.PackedLine.Estop[#MABS_ID] := #ReadMabsStatus.Estop;
	            DB_Global.Status.Line.PackedLine.Manual[#MABS_ID] := #ReadMabsStatus.Manual;
	            DB_Global.Status.Line.PackedLine.Stop[#MABS_ID] := #ReadMabsStatus.Stop;
	            DB_Global.Status.Line.PackedLine.Blockage[#MABS_ID] := #ReadMabsStatus.Blockage;
	        END_IF;
	        
	    END_REGION
	    
	    REGION Visu Color
	        
	        // each and every status of the conveyor will be mentioned by different colors in HMI panel
	        
	        #VisuColor.%X8 := #ReadMabsStatus.Blockage;
	        #VisuColor.%X0 := #ReadMabsStatus.ON;
	        #VisuColor.%X1 := #ReadMabsStatus.ReadytoRun;
	        #VisuColor.%X2 := #ReadMabsStatus.Occupied;
	        #VisuColor.%X3 := #ReadMabsStatus.Running;
	        #VisuColor.%X4 := #ReadMabsStatus.Fault;
	        #VisuColor.%X5 := #ReadMabsStatus.Estop;
	        #VisuColor.%X6 := #ReadMabsStatus.Manual;
	        #VisuColor.%X7 := #ReadMabsStatus.Stop;
	        
	        // convert word to Interger value: 
	        // color will be depends on the status priority (integer value) 
	        // reference: Conveyor image in HMI screen -> property -> Apperance   
	        
	        // ProductionLine
	        IF #Active.Line.ProductionLine THEN
	            DB_VisuColor.Line.ProductionLine.Conveyor[#MABS_ID] :=
	            WORD_TO_INT(#VisuColor);
	        END_IF;
	        // EmptyLine
	        IF #Active.Line.EmptyLine THEN
	            DB_VisuColor.Line.EmptyLine.Conveyor[#MABS_ID] :=
	            WORD_TO_INT(#VisuColor);
	        END_IF;
	        // PackedLine
	        IF #Active.Line.PackedLine THEN
	            DB_VisuColor.Line.PackedLine.Conveyor[#MABS_ID] :=
	            WORD_TO_INT(#VisuColor);
	        END_IF;
	        
	    END_REGION
	    
	END_REGION
	
	REGION Sorter sensor filter
	    
	    // cross sensor filter
	    #CROSS_SENSOR_FILTER(Sensor := #ReadInputSignal.CrossSensor,   ///#CrossSensor
	                         SensorFilterTime := #Parameter.CrossSensorFilterTime);
	    
	    
	END_REGION
	
	REGION MABS FUNCTIONALITY
	    
	    REGION rcv direction 
	        
	(*        // only if the mabs is not performing any operation
	        IF NOT #Upstream
	        THEN
	            #HoldSwing := TRUE;
	        ELSE
	            #HoldSwing := FALSE;
	        END_IF;
	        
	        IF NOT #HoldSwing THEN
	            
	            #Sort := #SortDir;
	            
	        END_IF; *)
	        
	        #Sort := #SortDir;
	        
	    END_REGION
	    
	    // Signal to RemoteIN1 / RemoteIN2 for specify swing direction and RemoteIN3 for swing must be 50ms or longer.
	    // Otherwise transfer ball may behaves unexpectedly.
	    // If the signal input of IN1 and IN2 (specifying the swing direction) is delayed from the signal input of IN3 (swing RUN),
	    // an unintended swing operation will occur.
	    // After outputting the swinging status, turn RemoteIN3 (Swing start) OFF.
	    
	    REGION MABS wheels
	        
	        // run mobs wheel 
	        // runs only when remoteIn3(swing) not active
	        
	        #mabs.Wheels := #UpstreamRunning;
	        
	    END_REGION
	    
	    // ==========================================================================================================================
	    // Swing status output
	    // ===================
	    
	    // SWING STATUS         RemoteOUT2  RemoteOUT3   Remark
	    // ------------         ----------  ----------   ------
	    // Straight (origin)        ON          ON       Outputs at the time when balls have been turned to the straight direction.
	    // Swing (CW)               ON          OFF      Outputs at the time when swing in CW direction is complete.
	    // Swing (CCW)              OFF         ON       Outputs at the time when swing in CCW direction is complete.
	    // Others                   OFF         OFF      During ball swing, when turning on power supply,
	    //                                               undetected swing position or occurring software error.
	    // ==========================================================================================================================                                              
	    
	    REGION Current position
	        
	        // current MABS position
	        
	        #CurrentPosition.left :=
	        NOT #RemoteOut2 AND
	        #RemoteOut3;
	        
	        #CurrentPosition.right :=
	        #RemoteOut2 AND
	        NOT #RemoteOut3;
	        
	        #CurrentPosition.straight :=
	        #RemoteOut2 AND
	        #RemoteOut3;
	        
	    END_REGION
	    
	    REGION HOMING
	        
	        // ==========================================================================================================================
	        // Initial operation (origin searching)
	        // ===================================
	        
	        #HomeCheckTimer.TON(IN := NOT #CurrentPosition.left AND
	                            NOT #CurrentPosition.right AND
	                            NOT #CurrentPosition.straight,
	                            PT := T#1s);
	        
	        #Home :=
	        NOT #HomeCheckTimer.Q;
	        
	        // home missing
	        
	        IF NOT #Home AND NOT #ReadMabsStatus.Stop THEN
	            #mabs.RemoteIn1 := TRUE;
	            #mabs.RemoteIn2 := TRUE;
	            #mabs.RemoteIn3 := TRUE;
	        END_IF;
	        
	    END_REGION
	    
	    // ==========================================================================================================================
	    // Specified swing direction
	    // =========================
	    
	    // SWING                                                    RemoteIN1  RemoteIN2   
	    // -----                                                    ---------  ---------   
	    // Divert direction to Straight direction (CW direction)       ON          ON       
	    // Divert direction to Straight direction (CCW direction)      ON          OFF      
	    // Straight direction to Divert direction (CW direction)       OFF         ON       
	    // Straight direction to Divert direction (CCW direction)      OFF         OFF                                                    .
	    // ==========================================================================================================================
	    // Start swinging
	    // ==============
	    
	    // swing    RemoteIN3
	    // -----    ---------  
	    // STOP         OFF
	    // RUN          ON  .
	    
	    // ==========================================================================================================================
	    
	    IF #ReadMabsStatus.ReadytoRun AND NOT #HoldFailure
	    THEN
	        
	        REGION swing delay
	            
	            #ToSt_DelayTimer(IN := #mabs.#RemoteIn1 AND #mabs.#RemoteIn2,
	                             PT := t#20ms,
	                             Q => #St_SwingDelay);
	            
	            #ToRt_DelayTimer(IN := NOT #mabs.#RemoteIn1 AND #mabs.#RemoteIn2,
	                             PT := t#20ms,
	                             Q => #Rt_SwingDelay);
	            
	            #ToLt_DelayTimer(IN := #mabs.#RemoteIn1 AND NOT #mabs.#RemoteIn2,
	                             PT := t#20ms,
	                             Q => #Lt_SwingDelay);
	            
	            // swing starts after few ms of turn decision made
	            IF (#St_SwingDelay OR
	                #Rt_SwingDelay OR
	                #Lt_SwingDelay) AND
	                NOT #noSwing
	            THEN
	                #mabs.RemoteIn3 := TRUE;
	            END_IF;
	            
	        END_REGION
	        
	        REGION Straight
	            
	            IF (#CurrentPosition.straight AND
	                #Sort.Straight) OR
	                (#CurrentPosition.right AND
	                #Sort.toRight) OR
	                (#CurrentPosition.left AND
	                #Sort.toLeft)
	            THEN
	                #mabs.RemoteIn3 := FALSE;
	                #noSwing := TRUE;
	            ELSE
	                #noSwing := FALSE;
	            END_IF;
	            
	            
	            // ================================================== ^^^
	            
	            // sort straight - actual position: right
	            
	            IF #Sort.Straight AND
	                NOT #CurrentPosition.straight AND
	                #CurrentPosition.right AND
	                NOT #CROSS_SENSOR_FILTER.FilteredSensor
	            THEN
	                #mabs.#RemoteIn1 := TRUE;
	                #mabs.RemoteIn2 := TRUE;
	            END_IF;
	            
	            // sort straight - actual position: left
	            
	            IF #Sort.Straight AND
	                NOT #CurrentPosition.straight AND
	                #CurrentPosition.left AND
	                NOT #CROSS_SENSOR_FILTER.FilteredSensor
	            THEN
	                #mabs.#RemoteIn1 := TRUE;
	                #mabs.RemoteIn2 := TRUE;
	            END_IF;
	            
	            // sort straight - actual position: straight
	            
	            IF #Sort.Straight AND
	                #CurrentPosition.straight AND
	                NOT #CurrentPosition.left AND
	                NOT #CurrentPosition.right AND
	                NOT #CROSS_SENSOR_FILTER.FilteredSensor
	            THEN
	                #mabs.RemoteIn3 := FALSE; // no swing
	            END_IF;
	            
	        END_REGION
	        
	        REGION to Right
	            
	            #RT_DelaySwing_toRight(CLK := #ToRt_DelayTimer.Q);
	            
	            // ================================================== >>>
	            
	            // sort right - actual position: straight/left
	            
	            IF #Sort.toRight AND
	                NOT #CurrentPosition.right AND
	                (#CurrentPosition.straight OR
	                #CurrentPosition.left) AND
	                NOT #CROSS_SENSOR_FILTER.FilteredSensor
	            THEN
	                #mabs.#RemoteIn1 := FALSE;
	                #mabs.RemoteIn2 := TRUE;
	            END_IF;
	            
	            // sort right - actual position: right
	            
	            IF #Sort.toRight AND
	                #CurrentPosition.right AND
	                NOT #CurrentPosition.left AND
	                NOT #CurrentPosition.straight AND
	                NOT #CROSS_SENSOR_FILTER.FilteredSensor
	            THEN
	                #mabs.RemoteIn3 := FALSE; // no swing
	            END_IF;
	            
	        END_REGION
	        
	        REGION to left
	            
	            #RT_DelaySwing_toLeft(CLK := #ToLt_DelayTimer.Q);
	            
	            // ================================================== <<<
	            
	            // sort left - actual position: straight/right
	            
	            IF #Sort.toLeft AND
	                NOT #CurrentPosition.left AND
	                (#CurrentPosition.straight OR
	                #CurrentPosition.right) AND
	                NOT #CROSS_SENSOR_FILTER.FilteredSensor
	            THEN
	                #mabs.#RemoteIn1 := FALSE;
	                #mabs.RemoteIn2 := TRUE;
	            END_IF;
	            
	            // sort left - actual position: left
	            
	            IF #Sort.toLeft AND
	                #CurrentPosition.left AND
	                NOT #CurrentPosition.straight AND
	                NOT #CurrentPosition.right AND
	                NOT #CROSS_SENSOR_FILTER.FilteredSensor
	            THEN
	                #mabs.RemoteIn3 := FALSE; // no swing
	            END_IF;
	            
	        END_REGION
	        
	        // ============================================================================================================
	        
	        #RemoteIn1 := #mabs.RemoteIn1;
	        #RemoteIn2 := #mabs.RemoteIn2;
	        #RemoteIn3 := #mabs.RemoteIn3;
	        
	        #RunWheels := #mabs.Wheels;
	        
	    END_IF;
	    
	    REGION Cmd excecution failure
	        
	        // if the cmd could not be excecuted, MABS getting program reset automatically
	        // Hold failure: makes all output to MABS value 0
	        // then starts executing cmd again
	        
	        IF #ReadMabsStatus.ReadytoRun AND #Home THEN
	            
	            // reset state change
	            #FT_Upstream(CLK := #Upstream);
	            #RT_DS_St(CLK := #Downstream_Straight);
	            #"RT_DS_Rt/Lt"(CLK := #"Downstream_Right/Left");
	            
	            // upstream not able to send tote in to MABS
	            #CmdExFailure.UpstreamCheckTimer(IN := #Upstream AND
	                                             ((NOT #Downstream_Straight AND #Sort.Straight) OR
	                                             (NOT #"Downstream_Right/Left" AND #Sort.toLeft)),
	                                             R := (#CmdExFailure.UpstreamCheckTimer.ET > t#30s) OR
	                                             #FT_Upstream.Q OR
	                                             #RT_DS_St.Q OR
	                                             #"RT_DS_Rt/Lt".Q OR
	                                             #SSR.ResetSystem,
	                                             PT := t#24h);
	            
	            // reset state change
	            #RT_ToStraight(CLK := #CurrentPosition.straight);
	            #RT_ToRight(CLK := #CurrentPosition.right);
	            #RT_ToLeft(CLK := #CurrentPosition.left);
	            #FT_Blockage(CLK := #ReadMabsStatus.Blockage);
	            
	            #CmdExFailure.Timer(IN := ((#Sort.Straight AND
	                                NOT #CurrentPosition.straight) OR
	                                (#Sort.toRight AND
	                                NOT #CurrentPosition.right) OR
	                                (#Sort.toLeft AND
	                                NOT #CurrentPosition.left)) OR
	                                #ReadMabsStatus.Blockage,
	                                R := (#CmdExFailure.Timer.ET > t#10s) OR
	                                #RT_ToStraight.Q OR
	                                #RT_ToRight.Q OR
	                                #RT_ToLeft.Q OR
	                                #FT_Blockage.Q OR
	                                #SSR.ResetSystem,
	                                PT := t#24h);
	            
	            #HoldFailure :=
	            ((#CmdExFailure.Timer.ET > t#5s) OR
	            (#CmdExFailure.UpstreamCheckTimer.ET > t#15s));
	            
	        END_IF;
	        
	        
	    END_REGION
	    
	    // stop if not ready
	    IF #Home AND (NOT #ReadMabsStatus.ReadytoRun OR #HoldFailure)
	    THEN
	        #RemoteIn1 := FALSE;
	        #RemoteIn2 := FALSE;
	        #RemoteIn3 := FALSE;
	        #RunWheels := FALSE;
	    END_IF;
	    
	    IF NOT #Home THEN
	        
	        #RemoteIn1 := #mabs.RemoteIn1;
	        #RemoteIn2 := #mabs.RemoteIn2;
	        #RemoteIn3 := #mabs.RemoteIn3;
	        
	    END_IF;
	    
	    
	END_REGION
	
	
	
END_FUNCTION_BLOCK
END_NAMESPACE

NAMESPACE Global
FUNCTION_BLOCK FB_MABS_Profinet
{ S7_Optimized_Access := 'TRUE' ; Published := 'TRUE' }
VERSION : 0.1
   VAR_INPUT 
      MABS_ID : Int;
      CrossSensor : Bool;
      Fault : Bool;
      UpstreamRunning : Bool;
      Downstream_Straight : Bool;
      "Downstream_Right/Left" : Bool;
      SortDir : ItemDir;
      ManIn : MABS_ManIn;
      Setpoints : MABS_Setpoint;
   END_VAR

   VAR_IN_OUT 
      MABS_IBP_in : IB_P01_02_03_in_64bytes_struct;
      MABS_IBP_out : IB_P01_02_03_out_64bytes_struct;
   END_VAR

   VAR 
      ReadInputSignal : Struct
         CrossSensor : Bool;
         EmergencyStop : Bool;
         Fault : Bool;
      END_STRUCT;
      Active : Struct
         Line : Struct
            ProductionLine : Bool;
            EmptyLine : Bool;
            PackedLine : Bool;
         END_STRUCT;
         EstopZone { S7_SetPoint := 'False'} : EsopZone;
      END_STRUCT;
      CROSS_SENSOR_FILTER : FB_Sensor;
      MABS_SENSOR_BLOCKAGE {InstructionName := 'IEC_TIMER'; LibVersion := '1.0'} : IEC_TIMER;
      MABS_STATUS_ON : FB_StatusON;
      MABS_STATUS_READY : FB_StatusReady;
      MABS_STATUS_FAULT : FB_StatusFault;
      AUTO_RESET : FB_AutoReset;
      MABS_CONTROL : FB_MABS_PNIO;
      SSR : SystemSSR;
      ReadMabsStatus : ConveyorStatus;
      ReadMabsParameter : ConveyorParameters := ((), [2(T#10ms)], (), (), (), ());
      MABSFault : Fault;
      SimuMode : Struct
         Sensor : Bool;
         Fault : Bool;
      END_STRUCT;
      StartUpTimer {InstructionName := 'TOF_TIME'; LibVersion := '1.0'; S7_SetPoint := 'False'} : TOF_TIME;
      FT_StartUp {InstructionName := 'F_TRIG'; LibVersion := '1.0'} : F_TRIG;
      SetStartUp { S7_SetPoint := 'True'} : Bool;
      VisuColor : Word;
      PhaseError : Bool;
      StartupMABS { S7_SetPoint := 'True'} : Bool;
      FilteredSensor { S7_SetPoint := 'True'} : Bool;
      AutoReset { S7_SetPoint := 'True'} : Bool;
      StopSystemFireActive : Bool;
      Sort { S7_SetPoint := 'False'} : ItemDir;
      Home : Bool;
      HomeCheckTimer {InstructionName := 'TON_TIME'; LibVersion := '1.0'} : TON_TIME;
      CurrentPosition : Struct
         left : Bool;
         right : Bool;
         straight : Bool;
      END_STRUCT;
      "Cmd+Setpoint" { ExternalAccessible := 'False'; ExternalVisible := 'False'; ExternalWritable := 'False'; S7_SetPoint := 'False'} : MABS;
   END_VAR


BEGIN
	// ==========================================================================================================================================
	// Company        : LogTech, s.r.o.
	// Created by     : Anton Vinoth Soundraraj
	// Block          : FB_MABS
	// Project        : Lékarna DC Chrudim
	// Project number : 23-157
	// ==========================================================================================================================================
	
	REGION Active Line
	    
	    // ProductionLine
	    IF (#MABS_ID >= _.gminProductionLine AND
	        #MABS_ID <= _.gmaxProductionLine)
	    THEN
	        #Active.Line.ProductionLine := TRUE;
	    END_IF;
	    
	    // EmptyLine
	    IF (#MABS_ID >= _.gminEmptyLine AND
	        #MABS_ID <= _.gmaxEmptyLine)
	    THEN
	        #Active.Line.EmptyLine := TRUE;
	    END_IF;
	    
	    // PackedLine
	    IF (#MABS_ID >= _.gminPackedLine AND
	        #MABS_ID <= _.gmaxPackedLine)
	    THEN
	        #Active.Line.PackedLine := TRUE;
	    END_IF;
	    
	END_REGION
	
	REGION Estop zone
	    
	    // Production Line A1
	    IF  (#MABS_ID >= _."gA1.6.1" AND
	        #MABS_ID <= _."gA1.6.2") OR
	        // Empty Line A1
	        (#MABS_ID >= _."gJ1.5.2" AND
	        #MABS_ID <= _."gJ1.6.2")
	    THEN
	        #Active.EstopZone."1" := TRUE;
	    END_IF;
	    
	    // Production Line A2
	    IF  (#MABS_ID >= _."gA1.9.1" AND
	        #MABS_ID <= _."gA1.9.2")
	    THEN
	        #Active.EstopZone."2" := TRUE;
	    END_IF;
	    
	END_REGION
	
	REGION SystemSSR
	    
	    //Zone 1
	    IF #Active.EstopZone."1" THEN
	        #SSR.StartSystem := DB_SystemSSR.Zone."1".StartSystem;
	        #SSR.StopSystem := DB_SystemSSR.Zone."1".StopSystem;
	        #SSR.ResetSystem := DB_SystemSSR.Zone."1".ResetSystem;
	    END_IF;
	    
	    //Zone 2
	    IF #Active.EstopZone."2" THEN
	        #SSR.StartSystem := DB_SystemSSR.Zone."2".StartSystem;
	        #SSR.StopSystem := DB_SystemSSR.Zone."2".StopSystem;
	        #SSR.ResetSystem := DB_SystemSSR.Zone."2".ResetSystem;
	    END_IF;
	    
	END_REGION
	
	REGION Read Simu inputs  
	    
	    // ProductionLine
	    IF #Active.Line.ProductionLine THEN
	        // read simu
	        #SimuMode.Sensor := DB_SystemSimu.TriggerSensor.Line.ProductionLine.Conveyor[#MABS_ID];
	        #SimuMode.Fault := DB_SystemSimu.TriggerFault.Line.ProductionLine.Conveyor[#MABS_ID];
	    END_IF;
	    
	    // EmptyLine
	    IF #Active.Line.EmptyLine THEN
	        // read simu
	        #SimuMode.Sensor := DB_SystemSimu.TriggerSensor.Line.EmptyLine.Conveyor[#MABS_ID];
	        #SimuMode.Fault := DB_SystemSimu.TriggerFault.Line.EmptyLine.Conveyor[#MABS_ID];
	    END_IF;
	    
	    // PackedLine
	    IF #Active.Line.PackedLine THEN
	        // read simu
	        #SimuMode.Sensor := DB_SystemSimu.TriggerSensor.Line.PackedLine.Conveyor[#MABS_ID];
	        #SimuMode.Fault := DB_SystemSimu.TriggerFault.Line.PackedLine.Conveyor[#MABS_ID];
	    END_IF;
	    
	END_REGION
	
	REGION Read Input
	    
	    // read all inputs to the block
	    // Conveyor input read signals
	    #ReadInputSignal.CrossSensor := #CrossSensor OR  // Not
	    #SimuMode.Sensor; // simu call
	    #ReadInputSignal.Fault := #Fault OR
	    #SimuMode.Fault; // simu call;
	    #ReadInputSignal.EmergencyStop := // all estop zones are connected together
	    _.DB_SafetyStandard.ToStandard.EstopActive;
	    
	END_REGION
	
	REGION READ AND INIT
	    
	    REGION parameters
	        
	        // ProductionLine
	        IF #Active.Line.ProductionLine THEN
	            #ReadMabsParameter := DB_ConveyorParameters.Line.ProductionLine.Conveyor[#MABS_ID];
	        END_IF;
	        // EmptyLine
	        IF #Active.Line.EmptyLine THEN
	            #ReadMabsParameter := DB_ConveyorParameters.Line.EmptyLine.Conveyor[#MABS_ID];
	        END_IF;
	        // PackedLine
	        IF #Active.Line.PackedLine THEN
	            #ReadMabsParameter := DB_ConveyorParameters.Line.PackedLine.Conveyor[#MABS_ID];
	        END_IF;
	        
	    END_REGION
	    
	    REGION FIRE
	        
	        // Fire signal from fire system stops the whole system
	        // System can be reset from Fire status only if the fire signal is deactivated
	        
	        // FIRE ALARM ACTIVE --> STOP SYSTEM
	        IF DB_SystemSimu.Fire THEN
	            #StopSystemFireActive := TRUE;
	        END_IF;
	        // RESET --> FIRE ALARM
	        IF #SSR.ResetSystem AND NOT DB_SystemSimu.Fire THEN
	            #StopSystemFireActive := FALSE;
	        END_IF;
	        
	    END_REGION
	    
	END_REGION
	
	REGION Conveyor startup
	    
	    // Conveyor StartUp: Conveyor startup signal after 5 second delay
	    
	    #StartUpTimer.TOF(IN := #SSR.StartSystem,
	                      PT := #ReadMabsParameter.StartUpTime);
	    
	    #FT_StartUp(CLK := #StartUpTimer.Q);
	    
	    // set startup after 5 seconds
	    #SetStartUp := #FT_StartUp.Q;
	    
	END_REGION
	
	REGION Conveyor Status
	    
	    REGION Status ON
	        
	        // ----------------------------------------->>>>>>> STATUS ON <<<<<<<-----------------------------------------
	        // FB_ConveyorStatusON
	        // called as IDMB
	        
	        #MABS_STATUS_ON(SystemStartActive := #SSR.StartSystem,
	                        StatusStop := #ReadMabsStatus.Stop,
	                        StatusEStop := #ReadMabsStatus.Estop,
	                        StatusManual := #ReadMabsStatus.Manual,
	                        StatusFault := #ReadMabsStatus.Fault,
	                        FireAlarmActive := #StopSystemFireActive,
	                        StatusON => #ReadMabsStatus.ON);
	        
	    END_REGION
	    
	    REGION Status Ready
	        
	        // ----------------------------------------->>>>>>> STATUS READY <<<<<<<-----------------------------------------
	        // FB_ConveyorStatusReady
	        // called as MIDB
	        
	        #MABS_STATUS_READY(StatusON := #ReadMabsStatus.ON,
	                           StatusESTOP := #ReadMabsStatus.Estop,
	                           StatusFAULT := #ReadMabsStatus.Fault,
	                           StatusMAN := #ReadMabsStatus.Manual,
	                           SignalFIRE := #StopSystemFireActive,
	                           SystemAlertTime := #ReadMabsParameter.StartUpTime,
	                           StatusReady => #ReadMabsStatus.ReadytoRun);
	        
	    END_REGION
	    
	    REGION Status Occupied
	        
	        // ----------------------------------------->>>>>>> STATUS OCCUPIED <<<<<<<-----------------------------------------
	        
	        #ReadMabsStatus.Occupied :=
	        #CROSS_SENSOR_FILTER.FilteredSensor;
	        
	    END_REGION
	    
	    REGION Status Running
	        
	        // ----------------------------------------->>>>>>> STATUS RUNNING <<<<<<<-----------------------------------------
	        
	        #ReadMabsStatus.Running :=
	        #ReadMabsStatus.ReadytoRun AND
	        #"Cmd+Setpoint".Run_balls;
	        
	    END_REGION
	    
	    REGION Status Fault
	        
	        // ----------------------------------------->>>>>>> STATUS FAULT <<<<<<<-----------------------------------------
	        
	        // Reading error signal from the motor drive
	        #MABSFault.Motor_Error := #ReadInputSignal.Fault;
	        
	        // FC_ConveyorStatusFault
	        #MABS_STATUS_FAULT(FaultActive := #MABSFault.Motor_Error,
	                           ResetFault := #SSR.ResetSystem,
	                           StatusRunning := #ReadMabsStatus.Running,
	                           FaultStatus => #ReadMabsStatus.Fault);
	        
	    END_REGION
	    
	    REGION Status ESTOP
	        
	        // ----------------------------------------->>>>>>> STATUS ESTOP <<<<<<<-----------------------------------------
	        
	        #AUTO_RESET(AckIN := #SSR.ResetSystem,
	                    Ack => #AutoReset);
	        
	        // EMERGENCY STOP ACTIVE --> STOP SYSTEM
	        IF #ReadInputSignal.EmergencyStop THEN
	            #ReadMabsStatus.Estop := TRUE;
	        END_IF;
	        // RESET --> EMERGENCY STOP
	        IF #AutoReset AND NOT #ReadInputSignal.EmergencyStop THEN
	            #ReadMabsStatus.Estop := FALSE;
	        END_IF;
	        
	    END_REGION
	    
	    REGION Status Stop
	        
	        // ----------------------------------------->>>>>>> STATUS STOP <<<<<<<-----------------------------------------
	        
	        IF #SSR.StopSystem THEN
	            #ReadMabsStatus.Stop := TRUE;
	        END_IF;
	        IF #SSR.StartSystem OR #SSR.ResetSystem THEN
	            #ReadMabsStatus.Stop := FALSE;
	        END_IF;
	        
	    END_REGION
	    
	    REGION Sensor Blockage
	        
	        // ----------------------------------------->>>>>>> STATUS BLOCKAGE <<<<<<<-------------------------------------
	        
	        // FB_SensorBlockage
	        // called as MIDB
	        
	        #MABS_SENSOR_BLOCKAGE.TON(IN := #ReadMabsStatus.ReadytoRun AND
	                                  #CROSS_SENSOR_FILTER.FilteredSensor,
	                                  PT := #ReadMabsParameter.SensorBlockageTime,
	                                  Q => #ReadMabsStatus.Blockage);
	        
	        // ==========================
	        // Sensor Blockage: HMI Alarm
	        // ==========================
	        // Sensor blockage alarm message is written to the first bit of the alarm word
	        // corresponding to the active line
	        
	        REGION alarm 
	            
	            // ==========================
	            // Sensor Blockage: HMI Alarm
	            // ==========================
	            // Sensor blockage alarm message is written to the alarm word
	            // corresponding to the active line
	            // ProductionLine
	            IF #Active.Line.ProductionLine THEN
	                DB_Alarm."word".Line.ProductionLine.Conveyor[#MABS_ID].%X0 := #ReadMabsStatus.Blockage;
	            END_IF;
	            // EmptyLine
	            IF #Active.Line.EmptyLine THEN
	               DB_Alarm."word".Line.EmptyLine.Conveyor[#MABS_ID].%X0 := #ReadMabsStatus.Blockage;
	            END_IF;
	            // PackedLine
	            IF #Active.Line.PackedLine THEN
	               DB_Alarm."word".Line.PackedLine.Conveyor[#MABS_ID].%X0 := #ReadMabsStatus.Blockage;
	            END_IF;
	            
	        END_REGION
	        
	    END_REGION
	    
	    REGION Visu Color
	        
	        // each and every status of the conveyor will be mentioned by different colors in HMI panel
	        
	        #VisuColor.%X8 := #ReadMabsStatus.Blockage;
	        #VisuColor.%X0 := #ReadMabsStatus.ON;
	        #VisuColor.%X1 := #ReadMabsStatus.ReadytoRun;
	        #VisuColor.%X2 := #ReadMabsStatus.Occupied;
	        #VisuColor.%X3 := #ReadMabsStatus.Running;
	        #VisuColor.%X4 := #ReadMabsStatus.Fault;
	        #VisuColor.%X5 := #ReadMabsStatus.Estop;
	        #VisuColor.%X6 := #ReadMabsStatus.Manual;
	        #VisuColor.%X7 := #ReadMabsStatus.Stop;
	        
	        // convert word to Interger value: 
	        // color will be depends on the status priority (integer value) 
	        // reference: Conveyor image in HMI screen -> property -> Apperance   
	        
	        // ProductionLine
	        IF #Active.Line.ProductionLine THEN
	            DB_VisuColor.Line.ProductionLine.Conveyor[#MABS_ID] :=
	            WORD_TO_INT(#VisuColor);
	        END_IF;
	        // EmptyLine
	        IF #Active.Line.EmptyLine THEN
	            DB_VisuColor.Line.EmptyLine.Conveyor[#MABS_ID] :=
	            WORD_TO_INT(#VisuColor);
	        END_IF;
	        // PackedLine
	        IF #Active.Line.PackedLine THEN
	            DB_VisuColor.Line.PackedLine.Conveyor[#MABS_ID] :=
	            WORD_TO_INT(#VisuColor);
	        END_IF;
	        
	    END_REGION
	    
	    REGION Global Status
	        
	        // write -> global status
	        // ProductionLine
	        IF #Active.Line.ProductionLine THEN
	            DB_Global.Status.Line.ProductionLine.On[#MABS_ID] := #ReadMabsStatus.ON;
	            DB_Global.Status.Line.ProductionLine.ReadyToRun[#MABS_ID] := #ReadMabsStatus.ReadytoRun;
	            DB_Global.Status.Line.ProductionLine.Occupied[#MABS_ID] := #ReadMabsStatus.Occupied;
	            DB_Global.Status.Line.ProductionLine.Running[#MABS_ID] := #ReadMabsStatus.Running;
	            DB_Global.Status.Line.ProductionLine.Fault[#MABS_ID] := #ReadMabsStatus.Fault;
	            DB_Global.Status.Line.ProductionLine.Estop[#MABS_ID] := #ReadMabsStatus.Estop;
	            DB_Global.Status.Line.ProductionLine.Manual[#MABS_ID] := #ReadMabsStatus.Manual;
	            DB_Global.Status.Line.ProductionLine.Stop[#MABS_ID] := #ReadMabsStatus.Stop;
	            DB_Global.Status.Line.ProductionLine.Blockage[#MABS_ID] := #ReadMabsStatus.Blockage;
	        END_IF;
	        // EmptyLine
	        IF #Active.Line.EmptyLine THEN
	            DB_Global.Status.Line.EmptyLine.On[#MABS_ID] := #ReadMabsStatus.ON;
	            DB_Global.Status.Line.EmptyLine.ReadyToRun[#MABS_ID] := #ReadMabsStatus.ReadytoRun;
	            DB_Global.Status.Line.EmptyLine.Occupied[#MABS_ID] := #ReadMabsStatus.Occupied;
	            DB_Global.Status.Line.EmptyLine.Running[#MABS_ID] := #ReadMabsStatus.Running;
	            DB_Global.Status.Line.EmptyLine.Fault[#MABS_ID] := #ReadMabsStatus.Fault;
	            DB_Global.Status.Line.EmptyLine.Estop[#MABS_ID] := #ReadMabsStatus.Estop;
	            DB_Global.Status.Line.EmptyLine.Manual[#MABS_ID] := #ReadMabsStatus.Manual;
	            DB_Global.Status.Line.EmptyLine.Stop[#MABS_ID] := #ReadMabsStatus.Stop;
	            DB_Global.Status.Line.EmptyLine.Blockage[#MABS_ID] := #ReadMabsStatus.Blockage;
	        END_IF;
	        // PackedLine
	        IF #Active.Line.PackedLine THEN
	            DB_Global.Status.Line.PackedLine.On[#MABS_ID] := #ReadMabsStatus.ON;
	            DB_Global.Status.Line.PackedLine.ReadyToRun[#MABS_ID] := #ReadMabsStatus.ReadytoRun;
	            DB_Global.Status.Line.PackedLine.Occupied[#MABS_ID] := #ReadMabsStatus.Occupied;
	            DB_Global.Status.Line.PackedLine.Running[#MABS_ID] := #ReadMabsStatus.Running;
	            DB_Global.Status.Line.PackedLine.Fault[#MABS_ID] := #ReadMabsStatus.Fault;
	            DB_Global.Status.Line.PackedLine.Estop[#MABS_ID] := #ReadMabsStatus.Estop;
	            DB_Global.Status.Line.PackedLine.Manual[#MABS_ID] := #ReadMabsStatus.Manual;
	            DB_Global.Status.Line.PackedLine.Stop[#MABS_ID] := #ReadMabsStatus.Stop;
	            DB_Global.Status.Line.PackedLine.Blockage[#MABS_ID] := #ReadMabsStatus.Blockage;
	        END_IF;
	        
	    END_REGION
	    
	END_REGION
	
	REGION Sorter sensor filter
	    
	    // cross sensor filter
	    #CROSS_SENSOR_FILTER(Sensor :=  #ReadInputSignal.CrossSensor,   ///#CrossSensor
	                         SensorFilterTime := #ReadMabsParameter.SensorFilterTime,
	                         FilteredSensor=> #FilteredSensor);
	    
	END_REGION
	
	REGION MABS LOGIC
	    
	    REGION rcv direction 
	        
	        IF NOT #FilteredSensor THEN
	            #Sort := #SortDir;
	        END_IF;
	        
	    END_REGION
	    
	    REGION MABS lib block
	        
	        #MABS_CONTROL(IBP_in  := #MABS_IBP_in,
	                      IBP_out := #MABS_IBP_out,
	                      MABS    := #"Cmd+Setpoint");
	        
	    END_REGION
	    
	    REGION run MABS wheels
	        
	        #"Cmd+Setpoint".Run_balls := #UpstreamRunning;
	        
	    END_REGION
	    
	    REGION Current position
	        
	        #CurrentPosition.left := #"Cmd+Setpoint".Left_Pos_reach;
	        #CurrentPosition.right := #"Cmd+Setpoint".Right_Pos_reach;
	        #CurrentPosition.straight := #"Cmd+Setpoint".Straight_Pos_reach;
	        
	    END_REGION
	    
	    REGION HOMING
	        
	        // ==========================================================================================================================
	        // Initial operation (home searching)
	        // ==================================
	        
	        // Home missing (if MABS could not receive any position in 't' duration)
	        #HomeCheckTimer.TON(IN := NOT #CurrentPosition.left AND
	                            NOT #CurrentPosition.right AND
	                            NOT #CurrentPosition.straight,
	                            PT := T#2s);
	        #Home :=
	        NOT #HomeCheckTimer.Q;
	        
	        // init HOME
	        IF NOT #Home AND NOT #ReadMabsStatus.Stop THEN
	            #"Cmd+Setpoint".Init := TRUE;
	        END_IF;
	        // RESET -> Init Home
	        IF #Home THEN
	            #"Cmd+Setpoint".Init := TRUE;
	        END_IF;
	        
	    END_REGION
	    
	    REGION Parameters
	        
	        // change balls direction
	        #"Cmd+Setpoint".Dir_balls := #Setpoints.ChangeBallsDirection;
	        // balls speed
	        #"Cmd+Setpoint".Speed_balls := #Setpoints.Speed_balls;
	        // offset for straight
	        #"Cmd+Setpoint".Init_offset := #Setpoints.Init_offset;
	        
	    END_REGION
	    
	    REGION Sorting logic
	        
	        IF #ReadMabsStatus.ReadytoRun
	        THEN
	            
	            REGION Straight
	                
	                // ================================================== ^^^
	                
	                // sort straight - actual position: right
	                
	                IF #Sort.Straight AND
	                    NOT #CurrentPosition.straight AND
	                    #CurrentPosition.right AND
	                    NOT #CROSS_SENSOR_FILTER.FilteredSensor
	                THEN
	                    #"Cmd+Setpoint".Switch_right_to_st := TRUE;
	                ELSE
	                    #"Cmd+Setpoint".Switch_right_to_st := FALSE;
	                END_IF;
	                
	                // sort straight - actual position: left
	                
	                IF #Sort.Straight AND
	                    NOT #CurrentPosition.straight AND
	                    #CurrentPosition.left AND
	                    NOT #CROSS_SENSOR_FILTER.FilteredSensor
	                THEN
	                    #"Cmd+Setpoint".Switch_left_to_st := TRUE;
	                ELSE
	                    #"Cmd+Setpoint".Switch_left_to_st := FALSE;
	                END_IF;
	                
	            END_REGION
	            
	            REGION to Right
	                
	                // ================================================== >>>
	                
	                // sort right - actual position: straight/left
	                
	                IF #Sort.toRight AND
	                    NOT #CurrentPosition.right AND
	                    (#CurrentPosition.straight OR
	                    #CurrentPosition.left) AND
	                    NOT #CROSS_SENSOR_FILTER.FilteredSensor
	                THEN
	                    #"Cmd+Setpoint".Switch_right := TRUE;
	                ELSE
	                    #"Cmd+Setpoint".Switch_right := FALSE;
	                END_IF;
	                
	            END_REGION
	            
	            REGION to left
	                
	                // ================================================== <<<
	                
	                // sort left - actual position: straight/right
	                
	                IF #Sort.toLeft AND
	                    NOT #CurrentPosition.left AND
	                    (#CurrentPosition.straight OR
	                    #CurrentPosition.right) AND
	                    NOT #CROSS_SENSOR_FILTER.FilteredSensor
	                THEN
	                    #"Cmd+Setpoint".Switch_left := TRUE;
	                ELSE
	                    #"Cmd+Setpoint".Switch_left := FALSE;
	                END_IF;
	                
	            END_REGION
	            
	            // ============================================================================================================
	            
	        END_IF;
	        
	    END_REGION
	    
	   REGION reset error 
	        
	        // reset error
	       IF #ReadMabsStatus.Fault AND
	           #SSR.ResetSystem
	       THEN
	            #"Cmd+Setpoint".Reset_error := TRUE;
	        ELSE
	            #"Cmd+Setpoint".Reset_error := FALSE;
	        END_IF;
	        
	    END_REGION
	    
	    REGION stop function
	        
	        // stop if not ready
	        IF NOT #ReadMabsStatus.ReadytoRun AND NOT #ReadMabsStatus.Manual
	        THEN
	            #"Cmd+Setpoint".Switch_left := FALSE;
	            #"Cmd+Setpoint".Switch_right := FALSE;
	            #"Cmd+Setpoint".Switch_right_to_st := FALSE;
	            #"Cmd+Setpoint".Switch_left_to_st := FALSE;
	        END_IF;
	        
	    END_REGION
	    
	END_REGION
	
	
	
END_FUNCTION_BLOCK
END_NAMESPACE

NAMESPACE Global
FUNCTION_BLOCK FB_S300_FullControl
{ S7_Optimized_Access := 'TRUE' ; Published := 'TRUE' }
VERSION : 0.1
   VAR_INPUT 
      TransferID : Int;
      TransferSensor : Bool;
      RollerUp : Bool;
      Fault : Bool;
      ReadyToRCV : Bool;
      UpstreamStraight : Bool;
      UpstreamArm : Bool;
      FrontSensor : Bool;
      EndSensor : Bool;
      "Left/RightSensor" : Bool;
      Downstream : Bool;
      PriorityStraight : Bool;
      PriorityArm : Bool;
   END_VAR

   VAR_OUTPUT 
      Direction : Bool;
      Cmd1 : Bool;
      Cmd2 : Bool;
      ErrorReset : Bool;
   END_VAR

   VAR 
      ReadInputSignal : Struct
         EmergencyStop : Bool;
         FireActive : Bool;
         Fault : Bool;
         TransferSensor : Bool;
      END_STRUCT;
      Active : Struct
         Line : Struct
            ProductionTotes : Bool;
         END_STRUCT;
         EstopZone { S7_SetPoint := 'False'} : EsopZone;
      END_STRUCT;
      TRANSFER_SENSOR : FB_Sensor;
      FRONT_SENSOR_FILTER : FB_Sensor;
      "Left/Right_SENSOR_FILTER" : FB_Sensor;
      End_Sensor_Filter : FB_Sensor;
      TRANSFER_SENSOR_BLOCKAGE {InstructionName := 'TON_TIME'; LibVersion := '1.0'} : TON_TIME;
      FRONT_SENSOR_BLOCKAGE {InstructionName := 'TON_TIME'; LibVersion := '1.0'} : TON_TIME;
      END_SENSOR_BLOCKAGE {InstructionName := 'TON_TIME'; LibVersion := '1.0'} : TON_TIME;
      "LEFT/RIGHT_SENSOR_BLOCKAGE" {InstructionName := 'TON_TIME'; LibVersion := '1.0'} : TON_TIME;
      TRANSFER_STATUS_ON : FB_StatusON;
      TRANSFER_STATUS_READY : FB_StatusReady;
      TRANSFER_STATUS_FAULT : FB_StatusFault;
      AUTO_RESET : FB_AutoReset;
      StartUpTimer {InstructionName := 'TOF_TIME'; LibVersion := '1.0'; S7_SetPoint := 'False'} : TOF_TIME;
      FT_StartUp {InstructionName := 'F_TRIG'; LibVersion := '1.0'} : F_TRIG;
      SetStartUp { S7_SetPoint := 'True'} : Bool;
      Init : Struct
         Line : Struct
            A1 : String := 'LineA1';
         END_STRUCT;
      END_STRUCT;
      SSR : SystemSSR;
      ReadTransferStatus : ConveyorStatus;
      ReadTransferParameters : ConveyorParameters_TransferUnit := ((), [2(T#10ms)], [2(T#10ms)], [2(T#10ms)], [()], (), (), ());
      ConveyorFault : Fault;
      StartupTransfer { S7_SetPoint := 'True'} : Bool;
      FilteredSensor { S7_SetPoint := 'True'} : Bool;
      StopSystemFireActive : Bool;
      ClearTransferArea : Bool;
      AutoReset : Bool;
      VisuColor : Word;
      Transfer : Struct
         ErrorReset : Bool;
         Direction : Bool;
         Command_1 : Bool;
         Command_2 : Bool;
      END_STRUCT;
      Intialization_PE {InstructionName := 'R_TRIG'; LibVersion := '1.0'; S7_SetPoint := 'False'} : R_TRIG;
      InitializationDone { S7_SetPoint := 'True'} : Bool;
      StartInitialization : Bool;
      ResetFault_PE {InstructionName := 'R_TRIG'; LibVersion := '1.0'} : R_TRIG;
   END_VAR


BEGIN
	// ==========================================================================================================================================
	// Company        : LogTech, s.r.o.
	// Created by     : Anton Vinoth Soundraraj
	// Block          : FB_S300_tTransMode
	// Project        : Lékarna DC Chrudim
	// Project number : 23-157
	// ==========================================================================================================================================
	
	REGION Active Line
	    
	        #Active.Line.ProductionTotes := TRUE;
	        
	    END_REGION
	    
	REGION Estop zone
	        
	        // Production Line A1
	    IF  #TransferID = _."gB1.6.1" 
	    THEN
	        #Active.EstopZone."1" := TRUE;
	    END_IF;
	        
	END_REGION
	    
	REGION SystemSSR
	        
	        //Zone 1
	        IF #Active.EstopZone."1" THEN
	            #SSR.StartSystem := DB_SystemSSR.Zone."1".StartSystem;
	            #SSR.StopSystem := DB_SystemSSR.Zone."1".StopSystem;
	            #SSR.ResetSystem := DB_SystemSSR.Zone."1".ResetSystem;
	        END_IF;
	        
	END_REGION
	    
	    
	
	REGION Initialization 
	    // Totes wait untill Initialization is done by haveing Rollers in High Postion
	    
	    #Intialization_PE(CLK := _.Global.DB_SystemSSR.Line.ProductionLine.StartSystem);
	    
	    IF #Intialization_PE.Q THEN
	        #StartInitialization := TRUE;
	    END_IF;
	    
	    IF #StartInitialization THEN
	        IF #RollerUp THEN
	            #InitializationDone := TRUE;
	            #StartInitialization := FALSE;
	        ELSE
	            #InitializationDone := FALSE;
	        END_IF;
	    END_IF;
	    
	END_REGION 
	
	REGION Read Input
	    
	    // read all inputs to the block
	    // Conveyor input read signals
	    #ReadInputSignal.TransferSensor := #TransferSensor;
	    #ReadInputSignal.Fault := #Fault;
	    // Read static tag connections
	    #ReadInputSignal.EmergencyStop := // all estop zones are connected together
	    _.DB_SafetyStandard.ToStandard.EstopActive;
	    // Common system input Read
	    #ReadInputSignal.FireActive :=
	    _.Global.DB_SystemSimu.Fire; // simu call
	    
	END_REGION
	
	REGION Conveyor startup
	    
	    // Conveyor StartUp: Conveyor startup signal after preset time
	    #StartUpTimer.TOF(IN := #SSR.StartSystem,
	                      PT := #ReadTransferParameters.StartUpTime);
	    
	    #FT_StartUp(CLK := #StartUpTimer.Q);
	    
	    // set startup after the preset
	    #SetStartUp := #FT_StartUp.Q;
	    
	END_REGION
	
	REGION READ AND INIT
	    
	    REGION Init conveyor parameters
	        
	        // Conveyor Parameter
	        // Line B1
	        IF #Active.Line.ProductionTotes THEN
	            #ReadTransferParameters := _.Global.DB_ConveyorParameters.Line.ProductionLine.TransferUnit[#TransferID];
	        END_IF;
	        
	    END_REGION
	    
	    REGION Sensor Filter
	        
	        // FB_Sensor
	        // called as MIDB
	        
	       #TRANSFER_SENSOR(Sensor := #ReadInputSignal.TransferSensor,
	                         SensorFilterTime := #ReadTransferParameters.SensorFilterTime,
	                         FilteredSensor => #FilteredSensor); 
	        
	        // front sensor filter
	        #FRONT_SENSOR_FILTER(Sensor := #FrontSensor,
	                             SensorFilterTime := #ReadTransferParameters.FrontSensorFilterTime);
	        
	        #"Left/Right_SENSOR_FILTER"(Sensor:=#"Left/RightSensor",
	                                    SensorFilterTime:=#ReadTransferParameters."Left/RightSensorFilterTime");
	        #End_Sensor_Filter(Sensor:=#EndSensor,
	                           SensorFilterTime:=#ReadTransferParameters.EndsensorFilterTime);
	        
	        
	    END_REGION
	    
	    REGION FIRE
	        
	        // Fire signal from fire system stops the whole system
	        // System can be reset from Fire status only if the fire signal is deactivated
	        
	        // FIRE ALARM ACTIVE --> STOP SYSTEM
	        IF #ReadInputSignal.FireActive THEN
	            #StopSystemFireActive := TRUE;
	        END_IF;
	        // RESET --> FIRE ALARM
	        IF #SSR.ResetSystem AND NOT #ReadInputSignal.FireActive THEN
	            #StopSystemFireActive := FALSE;
	        END_IF;
	        
	    END_REGION
	    
	END_REGION
	
	REGION Conveyor Status
	    
	    REGION Status ON
	        
	        // ----------------------------------------->>>>>>> STATUS ON <<<<<<<-----------------------------------------
	        // FB_ConveyorStatusON
	        // called as IDMB
	        
	        #TRANSFER_STATUS_ON(SystemStartActive := #SSR.StartSystem ,
	                            StatusStop := #ReadTransferStatus.Stop,
	                            StatusEStop := #ReadTransferStatus.Estop,
	                            StatusManual := #ReadTransferStatus.Manual,
	                            StatusFault := #ReadTransferStatus.Fault,
	                            FireAlarmActive := #StopSystemFireActive,
	                            StatusON => #ReadTransferStatus.ON);
	        
	    END_REGION
	    
	    REGION Status Ready
	        
	        // ----------------------------------------->>>>>>> STATUS READY <<<<<<<-----------------------------------------
	        // FB_ConveyorStatusReady
	        // called as MIDB
	        
	        #TRANSFER_STATUS_READY(StatusON := #ReadTransferStatus.ON, //AND #InitializationDone ,
	                               StatusESTOP := #ReadTransferStatus.Estop,
	                               StatusFAULT := #ReadTransferStatus.Fault,
	                               StatusMAN := #ReadTransferStatus.Manual,
	                               SignalFIRE := #StopSystemFireActive,
	                               SystemAlertTime := #ReadTransferParameters.StartUpTime,
	                               StatusReady => #ReadTransferStatus.ReadytoRun);
	        
	    END_REGION
	    
	    REGION Status Occupied
	        
	        // ----------------------------------------->>>>>>> STATUS OCCUPIED <<<<<<<-----------------------------------------
	        
	        #ReadTransferStatus.Occupied :=
	        #FilteredSensor AND
	        NOT #FRONT_SENSOR_FILTER.FilteredSensor AND 
	        NOT #"Left/Right_SENSOR_FILTER".FilteredSensor;
	        
	    END_REGION
	    
	    REGION Status Running
	        
	        // ----------------------------------------->>>>>>> STATUS RUNNING <<<<<<<-----------------------------------------
	        
	        #ReadTransferStatus.Running := #Transfer.Command_1 OR #Transfer.Command_2;
	        
	    END_REGION
	    
	    REGION Status Fault
	        
	        // Automatic reset trigger to the needed drive after wakeup from ESTOP power miss (only if needed)
	        // will trigger for every Reset active
	        
	        #AUTO_RESET(AckIN := #SSR.ResetSystem,
	                    Ack => #AutoReset);
	        
	        // ----------------------------------------->>>>>>> STATUS FAULT <<<<<<<-----------------------------------------
	        
	        #TRANSFER_STATUS_FAULT(FaultActive := #ReadInputSignal.Fault,
	                               ResetFault := #SSR.ResetSystem OR #AutoReset,
	                               StatusRunning := #ReadTransferStatus.Running,
	                               FaultStatus => #ReadTransferStatus.Fault);
	        
	        #ErrorReset := #SSR.ResetSystem AND #ReadTransferStatus.Fault;
	        
	    END_REGION
	    
	    REGION Status ESTOP
	        
	        // ----------------------------------------->>>>>>> STATUS ESTOP <<<<<<<-----------------------------------------
	        
	        // EMERGENCY STOP ACTIVE --> STOP SYSTEM
	        IF #ReadInputSignal.EmergencyStop THEN
	            #ReadTransferStatus.Estop := TRUE;
	        END_IF;
	        // RESET --> EMERGENCY STOP
	        IF #AutoReset AND NOT #ReadInputSignal.EmergencyStop THEN
	            #ReadTransferStatus.Estop := FALSE;
	        END_IF;
	        
	    END_REGION
	    
	    REGION Status Manual
	        
	        // ----------------------------------------->>>>>>> STATUS MANUAL <<<<<<<-----------------------------------------
	        
	        // Write to static from IO
	        // ACTIVATE --> MANUAL MODE
	        // Line B1
	        IF #Active.Line.ProductionTotes THEN
	            // SET --> MANUAL MODE
	            IF _.Global.DB_Manual.Line.ProductionLine.Conveyor[#TransferID].ManualEnable THEN
	                #ReadTransferStatus.Manual := TRUE;
	            END_IF;
	            // RESET --> MANUAL MODE
	            IF NOT _.Global.DB_Manual.Line.ProductionLine.Conveyor[#TransferID].ManualEnable AND #SSR.ResetSystem THEN
	                #ReadTransferStatus.Manual := FALSE;
	            END_IF;
	        END_IF;
	        
	    END_REGION
	    
	    REGION Status Stop
	        
	        // ----------------------------------------->>>>>>> STATUS STOP <<<<<<<-----------------------------------------
	        
	        IF #SSR.StopSystem THEN
	            #ReadTransferStatus.Stop := TRUE;
	        END_IF;
	        IF #SSR.StartSystem OR #SSR.ResetSystem THEN
	            #ReadTransferStatus.Stop := FALSE;
	        END_IF;
	        
	    END_REGION
	    
	    REGION Status Blockage
	        
	        // FB_SensorBlockage
	        // called as MIDB
	        #TRANSFER_SENSOR_BLOCKAGE(IN := #ReadTransferStatus.ReadytoRun AND #FilteredSensor AND NOT #Downstream,
	                                  PT := T#15s);
	        
	        #FRONT_SENSOR_BLOCKAGE(IN := #ReadTransferStatus.ReadytoRun AND #FrontSensor AND NOT #Downstream,
	                               PT := T#15s);
	        
	        #END_SENSOR_BLOCKAGE(IN := #ReadTransferStatus.ReadytoRun AND #EndSensor AND NOT #Downstream,
	                             PT := T#15s);
	        
	        #"LEFT/RIGHT_SENSOR_BLOCKAGE"(IN := #ReadTransferStatus.ReadytoRun AND #"Left/RightSensor" AND NOT #Downstream,
	                                      PT := T#5s);
	        
	        #ReadTransferStatus.Blockage :=
	        (#TRANSFER_SENSOR_BLOCKAGE.Q OR
	        #FRONT_SENSOR_BLOCKAGE.Q OR
	        #END_SENSOR_BLOCKAGE.Q OR
	        #"LEFT/RIGHT_SENSOR_BLOCKAGE".Q);
	        
	        // ==========================
	        // Sensor Blockage: HMI Alarm
	        // ==========================
	        // Sensor blockage alarm message is written to the alarm word
	        // corresponding to the active line
	        
	        REGION alarm 
	            
	            // ==========================
	            // Sensor Blockage: HMI Alarm
	            // ==========================
	            // Sensor blockage alarm message is written to the alarm word
	            // corresponding to the active line
	            // Line B1
	            IF #Active.Line.ProductionTotes THEN
	                _.Global.DB_Alarm."word".Line.ProductionLine.Conveyor[#TransferID].%X0 := #ReadTransferStatus.Blockage;
	            END_IF;
	            
	        END_REGION
	        
	    END_REGION
	    
	    REGION Visu Color
	        
	        // each and every status of the conveyor will be mentioned by different colors in HMI panel
	        
	        #VisuColor.%X8 := #ReadTransferStatus.Blockage;
	        #VisuColor.%X0 := #ReadTransferStatus.ON;
	        #VisuColor.%X1 := #ReadTransferStatus.ReadytoRun;
	        #VisuColor.%X2 := #ReadTransferStatus.Occupied;
	        #VisuColor.%X3 := #ReadTransferStatus.Running;
	        #VisuColor.%X4 := #ReadTransferStatus.Fault;
	        #VisuColor.%X5 := #ReadTransferStatus.Estop;
	        #VisuColor.%X6 := #ReadTransferStatus.Manual;
	        #VisuColor.%X7 := #ReadTransferStatus.Stop;
	        
	        // convert word to Interger value: 
	        // color will be depends on the status priority (integer value) 
	        // reference: Conveyor image in HMI screen -> property -> Apperance   
	        
	        // Line B1
	        IF #Active.Line.ProductionTotes THEN
	            _.Global.DB_VisuColor.Line.ProductionLine.Conveyor[#TransferID] :=
	            WORD_TO_INT(#VisuColor);
	        END_IF;
	        
	    END_REGION
	    
	    REGION Global Status
	        
	        // write -> global status
	        // Line B1
	        IF #Active.Line.ProductionTotes THEN
	            _.Global.DB_Global.Status.Line.ProductionLine.On[#TransferID] := #ReadTransferStatus.ON;
	            _.Global.DB_Global.Status.Line.ProductionLine.ReadyToRun[#TransferID] := #ReadTransferStatus.ReadytoRun;
	            _.Global.DB_Global.Status.Line.ProductionLine.Occupied[#TransferID] := #ReadTransferStatus.Occupied;
	            _.Global.DB_Global.Status.Line.ProductionLine.Running[#TransferID] := #ReadTransferStatus.Running;
	            _.Global.DB_Global.Status.Line.ProductionLine.Fault[#TransferID] := #ReadTransferStatus.Fault;
	            _.Global.DB_Global.Status.Line.ProductionLine.Estop[#TransferID] := #ReadTransferStatus.Estop;
	            _.Global.DB_Global.Status.Line.ProductionLine.Manual[#TransferID] := #ReadTransferStatus.Manual;
	            _.Global.DB_Global.Status.Line.ProductionLine.Stop[#TransferID] := #ReadTransferStatus.Stop;
	            _.Global.DB_Global.Status.Line.ProductionLine.Blockage[#TransferID] := #ReadTransferStatus.Blockage;
	        END_IF;
	        
	    END_REGION
	    
	END_REGION
	
	//===================
	//Transfer Logic
	//===================
	
	REGION #Transfer Logic
	    IF #ReadTransferStatus.ReadytoRun THEN
	        REGION Belt Infeed/Outfeed
	            
	            REGION Belt UP
	                
	                IF (#UpstreamStraight AND
	                    #PriorityStraight AND
	                    NOT #PriorityArm AND
	                    NOT #ReadTransferStatus.Occupied) AND
	                    #RollerUp OR
	                    (#ReadTransferStatus.Occupied AND
	                    #RollerUp)
	                THEN
	                    #Transfer.Command_1 := TRUE;  //Input signal Command 1
	                    #Transfer.Command_2 := TRUE;  //Input signal Command 2
	                    #Transfer.Direction := TRUE;  // Input signal direction of rotation
	                END_IF;
	                
	            END_REGION
	            
	            REGION Belt Run
	                // Run Belt until the negative edge of Sensor
	                
	                IF NOT #RollerUp AND
	                    (#UpstreamStraight OR
	                    #FRONT_SENSOR_FILTER.FilteredSensor) AND
	                    #PriorityStraight AND
	                    NOT #PriorityArm AND
	                    NOT #ReadTransferStatus.Occupied OR
	                    (#ReadTransferStatus.Occupied AND
	                    NOT #RollerUp)
	                THEN
	                    #Transfer.Command_1 := TRUE;  //Input signal Command 1
	                    #Transfer.Command_2 := FALSE;  //Input signal Command 2
	                    #Transfer.Direction := DB_S300SetPoint.Line.ProductionLine.DirChange.Conveyor[#TransferID].BeltDir;  // Input signal direction of rotation
	                END_IF;
	                
	            END_REGION
	            
	            
	        END_REGION
	        
	        REGION Roller Infeed Belt OutFeed
	            REGION Roller Up
	                IF #UpstreamArm AND
	                    #PriorityArm AND
	                    NOT #PriorityStraight AND
	                    NOT #ReadTransferStatus.Occupied AND
	                    NOT #RollerUp 
	                THEN
	                    #Transfer.Command_1 := TRUE;  //Input signal Command 1
	                    #Transfer.Command_2 := TRUE;  //Input signal Command 2
	                    #Transfer.Direction := FALSE;  // Input signal direction of rotation
	                END_IF;
	                
	            END_REGION
	            
	            REGION Roller Run
	                //Run the roller until you get negative edge of Left/Right sensor
	                IF (#UpstreamArm OR
	                    #"Left/Right_SENSOR_FILTER".FilteredSensor) AND
	                    #PriorityArm AND
	                    NOT #PriorityStraight AND
	                    NOT #ReadTransferStatus.Occupied AND
	                    #RollerUp 
	                THEN
	                    #Transfer.Command_1 := FALSE;  //Input signal Command 1
	                    #Transfer.Command_2 := TRUE;  //Input signal Command 2
	                    #Transfer.Direction := DB_S300SetPoint.Line.ProductionLine.DirChange.Conveyor[#TransferID].RollerDir;  // Input signal direction of rotation
	                END_IF;
	                
	            END_REGION
	            
	        END_REGION
	        
	    END_IF;
	    
	    REGION TRANSFER OFF
	        
	        IF  NOT #ReadTransferStatus.ReadytoRun OR 
	            (#ReadTransferStatus.Occupied AND
	            #Downstream) OR
	            (NOT #ReadTransferStatus.Occupied AND
	            NOT #End_Sensor_Filter.FilteredSensor AND
	            NOT #FRONT_SENSOR_FILTER.FilteredSensor AND
	            NOT #"Left/Right_SENSOR_FILTER".FilteredSensor AND 
	            NOT #UpstreamArm AND
	            NOT #UpstreamStraight)
	        THEN
	            #Transfer.Command_1 := FALSE;
	            #Transfer.Command_2 := FALSE;
	        END_IF;
	        
	    END_REGION
	    
	    REGION Write output
	        
	        // Static to output
	        
	        #Direction := #Transfer.Direction;
	        #Cmd1 := #Transfer.Command_1;
	        #Cmd2 := #Transfer.Command_2;
	        #ErrorReset := #Transfer.ErrorReset;
	        
	    END_REGION
	    
	    REGION Reset Fault 
	        (* #ResetFault_PE(CLK:=#Fault);
	        
	        IF #ResetFault_PE.Q THEN
	            #ErrorReset := TRUE;
	        END_IF; *)
	        
	        #ErrorReset := #SSR.ResetSystem;
	        
	    END_REGION 
	    
	    
	END_REGION
	
	
END_FUNCTION_BLOCK
END_NAMESPACE

NAMESPACE Global
FUNCTION_BLOCK FB_S300_tTransMode
{ S7_Optimized_Access := 'TRUE' ; Published := 'TRUE' }
VERSION : 0.1
   VAR_INPUT 
      TransferID : Int;
      TransferSensor : Bool;
      Fault : Bool;
      ReadyToRCV : Bool;
      Upstream : Bool;
      FrontSensor : Bool;
      EndSensor : Bool;
      "Left/RightSensor" : Bool;
      Downstream : Bool;
      FrontSensorFilterTime : Array[1..2] of Time;
      TransferDirection : ItemDir;
   END_VAR

   VAR_OUTPUT 
      StartSignal : Bool;
      Cmd1 : Bool;
      Cmd2 : Bool;
      ErrorReset : Bool;
   END_VAR

   VAR 
      ReadInputSignal : Struct
         EmergencyStop : Bool;
         FireActive : Bool;
         Fault : Bool;
         TransferSensor : Bool;
      END_STRUCT;
      Active : Struct
         Line : Struct
            ProductionLine : Bool;
            EmptyLine : Bool;
            PackedLine : Bool;
         END_STRUCT;
         EstopZone { S7_SetPoint := 'False'} : EsopZone;
      END_STRUCT;
      TRANSFER_SENSOR : FB_Sensor;
      FRONT_SENSOR_FILTER : FB_Sensor;
      TRANSFER_SENSOR_BLOCKAGE {InstructionName := 'TON_TIME'; LibVersion := '1.0'} : TON_TIME;
      FRONT_SENSOR_BLOCKAGE {InstructionName := 'TON_TIME'; LibVersion := '1.0'} : TON_TIME;
      END_SENSOR_BLOCKAGE {InstructionName := 'TON_TIME'; LibVersion := '1.0'} : TON_TIME;
      "LEFT/RIGHT_SENSOR_BLOCKAGE" {InstructionName := 'TON_TIME'; LibVersion := '1.0'} : TON_TIME;
      TRANSFER_STATUS_ON : FB_StatusON;
      TRANSFER_STATUS_READY : FB_StatusReady;
      TRANSFER_STATUS_FAULT : FB_StatusFault;
      AUTO_RESET : FB_AutoReset;
      StartUpTimer {InstructionName := 'TOF_TIME'; LibVersion := '1.0'; S7_SetPoint := 'False'} : TOF_TIME;
      FT_StartUp {InstructionName := 'F_TRIG'; LibVersion := '1.0'} : F_TRIG;
      SetStartUp { S7_SetPoint := 'True'} : Bool;
      Init : Struct
         Line : Struct
            A1 : String := 'LineA1';
         END_STRUCT;
      END_STRUCT;
      SSR : SystemSSR;
      ReadTransferStatus : ConveyorStatus;
      ReadTransferParameters : ConveyorParameters := ((), [2(T#10ms)], (), (), (), ());
      ConveyorFault : Fault;
      StartupTransfer { S7_SetPoint := 'True'} : Bool;
      FilteredSensor { S7_SetPoint := 'True'} : Bool;
      StopSystemFireActive : Bool;
      ClearTransferArea : Bool;
      AutoReset : Bool;
      VisuColor : Word;
      Transfer : Struct
         RcvInfeed : Bool;
         StartSignal : Bool;
         Command_1 : Bool;
         Command_2 : Bool;
      END_STRUCT;
      NegEdgeUpstream {InstructionName := 'F_TRIG'; LibVersion := '1.0'; S7_SetPoint := 'False'} : F_TRIG;
      CrossSensorFilterTime { S7_SetPoint := 'True'} : Array[0..1] of Time;
      sTransferDirection { S7_SetPoint := 'False'} : ItemDir;
      SimuMode : Struct
         Sensor : Bool;
         Fault : Bool;
      END_STRUCT;
   END_VAR


BEGIN
	// ==========================================================================================================================================
	// Company        : LogTech, s.r.o.
	// Created by     : Anton Vinoth Soundraraj
	// Block          : FB_S300_tTransMode
	// Project        : Lékarna DC Chrudim
	// Project number : 23-157
	// ==========================================================================================================================================
	
	REGION Active Line
	    
	    // ProductionLine
	    IF (#TransferID >= _.gminProductionLine AND
	        #TransferID <= _.gmaxProductionLine)
	    THEN
	        #Active.Line.ProductionLine := TRUE;
	    END_IF;
	    
	    // EmptyLine
	    IF (#TransferID >= _.gminEmptyLine AND
	        #TransferID <= _.gmaxEmptyLine)
	    THEN
	        #Active.Line.EmptyLine := TRUE;
	    END_IF;
	    
	    // PackedLine
	    IF (#TransferID >= _.gminPackedLine AND
	        #TransferID <= _.gmaxPackedLine)
	    THEN
	        #Active.Line.PackedLine := TRUE;
	    END_IF;
	    
	END_REGION
	
	REGION Estop zone
	    
	    // Production Line A1
	    IF  (#TransferID >= _."gB1.6.1" AND
	        #TransferID <= _."gC1.3.1")
	    THEN
	        #Active.EstopZone."1" := TRUE;
	    END_IF;
	    
	    // Production Line A2
	    IF  (#TransferID >= _."gA1.13.1" AND
	        #TransferID <= _."gA2.1.1") OR
	        (#TransferID >= _."gD1.9.1" AND
	        #TransferID <= _."gD1.10.1") 
	    THEN
	        #Active.EstopZone."2" := TRUE;
	    END_IF;
	    
	END_REGION
	
	REGION SystemSSR
	    
	    //Zone 1
	    IF #Active.EstopZone."1" THEN
	        #SSR.StartSystem := DB_SystemSSR.Zone."1".StartSystem;
	        #SSR.StopSystem := DB_SystemSSR.Zone."1".StopSystem;
	        #SSR.ResetSystem := DB_SystemSSR.Zone."1".ResetSystem;
	    END_IF;
	    
	    //Zone 2
	    IF #Active.EstopZone."2" THEN
	        #SSR.StartSystem := DB_SystemSSR.Zone."2".StartSystem;
	        #SSR.StopSystem := DB_SystemSSR.Zone."2".StopSystem;
	        #SSR.ResetSystem := DB_SystemSSR.Zone."2".ResetSystem;
	    END_IF;
	    
	END_REGION
	
	REGION Read Simu inputs  
	    
	    // ProductionLine
	    IF #Active.Line.ProductionLine THEN
	        // read simu
	        #SimuMode.Sensor := DB_SystemSimu.TriggerSensor.Line.ProductionLine.Conveyor[#TransferID];
	        #SimuMode.Fault := DB_SystemSimu.TriggerFault.Line.ProductionLine.Conveyor[#TransferID];
	    END_IF;
	    
	    // EmptyLine
	    IF #Active.Line.EmptyLine THEN
	        // read simu
	        #SimuMode.Sensor := DB_SystemSimu.TriggerSensor.Line.EmptyLine.Conveyor[#TransferID];
	        #SimuMode.Fault := DB_SystemSimu.TriggerFault.Line.EmptyLine.Conveyor[#TransferID];
	    END_IF;
	    
	    // PackedLine
	    IF #Active.Line.PackedLine THEN
	        // read simu
	        #SimuMode.Sensor := DB_SystemSimu.TriggerSensor.Line.PackedLine.Conveyor[#TransferID];
	        #SimuMode.Fault := DB_SystemSimu.TriggerFault.Line.PackedLine.Conveyor[#TransferID];
	    END_IF;
	    
	END_REGION
	
	REGION Read Input
	    
	    // read all inputs to the block
	    // Conveyor input read signals
	    #ReadInputSignal.TransferSensor := #TransferSensor OR  #SimuMode.Sensor; // simu call;
	    #ReadInputSignal.Fault := #Fault OR #SimuMode.Fault;
	    // Read static tag connections
	    #ReadInputSignal.EmergencyStop := // all estop zones are connected together
	    _.DB_SafetyStandard.ToStandard.EstopActive;
	    // Common system input Read
	    #ReadInputSignal.FireActive :=
	    DB_SystemSimu.Fire; // simu call
	    
	END_REGION
	
	REGION Conveyor startup
	    
	    // Conveyor StartUp: Conveyor startup signal after preset time
	    #StartUpTimer.TOF(IN := #SSR.StartSystem,
	                      PT := #ReadTransferParameters.StartUpTime);
	    
	    #FT_StartUp(CLK := #StartUpTimer.Q);
	    
	    // set startup after the preset
	    #SetStartUp := #FT_StartUp.Q;
	    
	END_REGION
	
